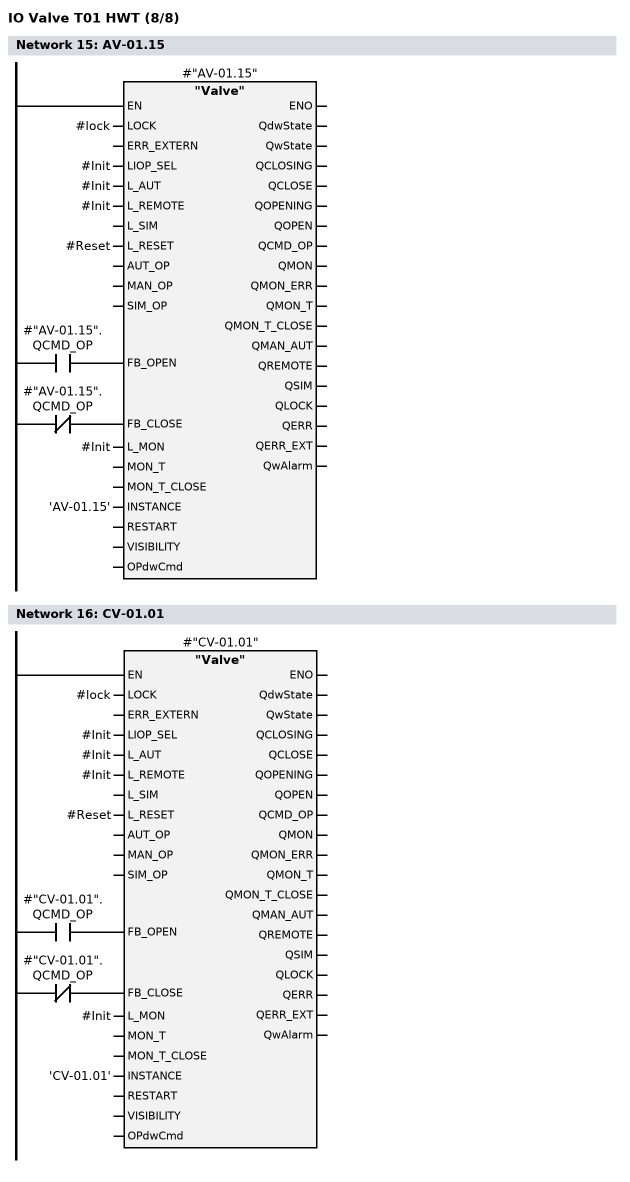
   RUNG wire#powerrail
      #"AV-01.15"(FB_OPEN := wire#w1, FB_CLOSE := wire#w2, LOCK := #lock, ERR_EXTERN :=, LIOP_SEL := #Init, L_AUT := #Init, L_REMOTE := #Init, L_SIM :=, L_RESET := #Reset, AUT_OP :=, MAN_OP :=, SIM_OP :=, L_MON := #Init, MON_T :=, MON_T_CLOSE :=, INSTANCE := 'AV-01.15', RESTART :=, VISIBILITY :=, OPdwCmd :=, QdwState =>, QwState =>, QCLOSING =>, QCLOSE =>, QOPENING =>, QOPEN =>, QCMD_OP =>, QMON =>, QMON_ERR =>, QMON_T =>, QMON_T_CLOSE =>, QMAN_AUT =>, QREMOTE =>, QSIM =>, QLOCK =>, QERR =>, QERR_EXT =>, QwAlarm =>)
   END_RUNG
   RUNG wire#powerrail
      Contact( #"AV-01.15".QCMD_OP )
   END_RUNG wire#w1
   RUNG wire#powerrail
      I_Contact( #"AV-01.15".QCMD_OP )
   END_RUNG wire#w2
   // the same network as SCL:
   #"AV-01.15"(LOCK := #lock,   // "Valve"
               LIOP_SEL := #Init,
               L_AUT := #Init,
               L_REMOTE := #Init,
               L_RESET := #Reset,
               FB_OPEN := #"AV-01.15".QCMD_OP,
               FB_CLOSE := NOT #"AV-01.15".QCMD_OP,
               L_MON := #Init,
               INSTANCE := 'AV-01.15');
END_REGION

REGION Network 16: CV-01.01
   RUNG wire#powerrail
      #"CV-01.01"(FB_OPEN := wire#w1, FB_CLOSE := wire#w2, LOCK := #lock, ERR_EXTERN :=, LIOP_SEL := #Init, L_AUT := #Init, L_REMOTE := #Init, L_SIM :=, L_RESET := #Reset, AUT_OP :=, MAN_OP :=, SIM_OP :=, L_MON := #Init, MON_T :=, MON_T_CLOSE :=, INSTANCE := 'CV-01.01', RESTART :=, VISIBILITY :=, OPdwCmd :=, QdwState =>, QwState =>, QCLOSING =>, QCLOSE =>, QOPENING =>, QOPEN =>, QCMD_OP =>, QMON =>, QMON_ERR =>, QMON_T =>, QMON_T_CLOSE =>, QMAN_AUT =>, QREMOTE =>, QSIM =>, QLOCK =>, QERR =>, QERR_EXT =>, QwAlarm =>)
   END_RUNG
   RUNG wire#powerrail
      Contact( #"CV-01.01".QCMD_OP )
   END_RUNG wire#w1
   RUNG wire#powerrail
      I_Contact( #"CV-01.01".QCMD_OP )
   END_RUNG wire#w2
   // the same network as SCL:
   #"CV-01.01"(LOCK := #lock,   // "Valve"
               LIOP_SEL := #Init,
               L_AUT := #Init,
               L_REMOTE := #Init,
               L_RESET := #Reset,
               FB_OPEN := #"CV-01.01".QCMD_OP,
               FB_CLOSE := NOT #"CV-01.01".QCMD_OP,
               L_MON := #Init,
               INSTANCE := 'CV-01.01');
END_REGION
END_FUNCTION_BLOCK

FUNCTION_BLOCK "BLEND"   // FB16, LAD
{ S7_Optimized_Access := 'FALSE' }
VERSION : 0.1
// stored: AutoNumber true, IsIECCheckEnabled false, SetENOAutomatically false, UDAEnableTagReadback false
   VAR_INPUT
      Lock : Bool := true;
      Reset : Bool;
      ENTransfer : Bool;
      ENProd : Bool;
      THE_ProdReq : Bool;   // THE Product Request
      THE_ProdLineOpen : Bool;   // THE Line Transfer Open
      THE_CIPLineOpen : Bool;   // THE CIP Line Open
      THE_CIP_En : Bool;   // THE CIP Enable
      MixproofFlip : Bool;
      FB_AV_Transfer : Bool;
      FB_P_Transfer : Bool;
      Level : Real;   // Tank Level Transmitter
      Temp : Real;   // Tank Temp Transmitter
      TransfPump_AVSpeed : Real;
   END_VAR
   VAR_OUTPUT
      Q_Prod : Bool;   // Product Available
      Q_Trans : Bool;   // Transfer to Mix in Progress
      Q_CIPReq : Bool;   // CIP Request
      Q_MixProofFlif : Bool;   // Mixproof Valve Flip
      QAV_Transfer : Bool;
      QP_Transfer : Bool;
   END_VAR
   VAR DB_SPECIFIC
      Cmd : Struct
         Transfer_ON : Bool;
         Transfer_OFF : Bool;
      END_STRUCT;
      HMI : Struct
         Cmd : DWord;
         Cmd_EN : DWord;
         Cmd_Stat : DWord;
         MatSel : DWord;
         DoseStart : DWord;
         DosePause : DWord;
         DoseStop : DWord;
         DoseState : DWord;
      END_STRUCT;
      Tank_Par : Struct
         LL : Real := 2.0;   // Tank Low Level
         LB_OFF : Real := 17.0;
         LB_ON : Real := 20.0;
         LB1_OFF : Real := 10.0;   // Level Under Lower Blade
         LB1_ON : Real := 15.0;   // Level Over Lower Blade
         LB2_OFF : Real := 30.0;   // Level Under Medium Blade
         LB2_ON : Real := 35.0;   // Level Over Medium Blade
         LB3_OFF : Real := 60.0;   // Level Under Upper Blade
         LB3_ON : Real := 65.0;   // Level Over Upper Blade
         P01_ProdSP : Real := 5.0;   // Transfer pump Setpoint speed at product transfer
         P01_CIPSP : Real := 50.0;   // Transfer pump Setpoint speed at CIP
      END_STRUCT;
      Tank_Sta : Struct   // Tank Low Level
         LL : Bool;   // Level Under Lower Blade
         LB_OFF : Bool;
         LB_ON : Bool;
         LB1_OFF : Bool;   // Level Over Lower Blade
         LB1_ON : Bool;   // Level Under Medium Blade
         LB2_OFF : Bool;   // Level Over Medium Blade
         LB2_ON : Bool;   // Level Under Upper Blade
         LB3_OFF : Bool;   // Level Over Upper Blade
         LB3_ON : Bool;
         Agi_ON : Bool;
         TranferON : Bool;
         Inload : Bool;
         CIPRequest : Bool;
         AwysON : Bool;
      END_STRUCT;
   END_VAR
   VAR
      SP_Water : "RawDose";
      SP_Sugar { S7_SetPoint := 'True'} : "RawDose";
      SP_Garam { S7_SetPoint := 'True'} : "RawDose";
      SP_ChiliAwet_1 { S7_SetPoint := 'True'} : "RawDose";
      SP_ChiliAwet_2 { S7_SetPoint := 'True'} : "RawDose";
      SP_ChiliAwet_3 { S7_SetPoint := 'True'} : "RawDose";
      SP_ChiliFresh_1 { S7_SetPoint := 'True'} : "RawDose";
      SP_ChiliFresh_2 { S7_SetPoint := 'True'} : "RawDose";
      SP_ChiliFresh_3 { S7_SetPoint := 'True'} : "RawDose";
      SP_Garlic { S7_SetPoint := 'True'} : "RawDose";
      SP_Vinegar { S7_SetPoint := 'True'} : "RawDose";
      SP_Tomato { S7_SetPoint := 'True'} : "RawDose";
      SP_Homomix { S7_SetPoint := 'True'} : "RawDose";
      SP_Rework { S7_SetPoint := 'True'} : "RawDose";
      Water : "DOSE";
      Sugar { S7_SetPoint := 'True'} : "DOSE";
      Garam : "DOSE";
      ChiliAwet_1 { S7_SetPoint := 'True'} : "DOSE";
      ChiliAwet_2 { S7_SetPoint := 'True'} : "DOSE";
      ChiliAwet_3 { S7_SetPoint := 'True'} : "DOSE";
      ChiliFresh_1 { S7_SetPoint := 'True'} : "DOSE";
      ChiliFresh_2 { S7_SetPoint := 'True'} : "DOSE";
      ChiliFresh_3 { S7_SetPoint := 'True'} : "DOSE";
      Garlic { S7_SetPoint := 'True'} : "DOSE";
      Vinegar { S7_SetPoint := 'True'} : "DOSE";
      Tomato { S7_SetPoint := 'True'} : "DOSE";
      Homomix { S7_SetPoint := 'True'} : "DOSE";
      Rework { S7_SetPoint := 'True'} : "DOSE";
   END_VAR
   VAR DB_SPECIFIC
      RdyforTransfer : Struct
         cmd_on : Bool;
         cmd_off : Bool;
         EnCmd : Bool;
         Stat_ON : Bool;
         Stat_Stop : Bool;
      END_STRUCT;
      Transfer : Struct
         cmd_on : Bool;
         cmd_off : Bool;
         EnCmd : Bool;
         Stat_ON : Bool;
         Stat_Stop : Bool;
      END_STRUCT;
      CIP : Struct
         cmd_on : Bool;
         cmd_off : Bool;
         EnCmd : Bool;
         Stat_ON : Bool;
         Stat_Stop : Bool;
      END_STRUCT;
      Agitator : Struct
         cmd_on : Bool;
         cmd_off : Bool;
         EnCmd : Bool;
         Stat_ON : Bool;
         Stat_Stop : Bool;
      END_STRUCT;
      PumpOFFTimer : TON_TIME;
      TransitionTimer { S7_SetPoint := 'True'} : TON_TIME;
   END_VAR
BEGIN

REGION Network 1: Always ON
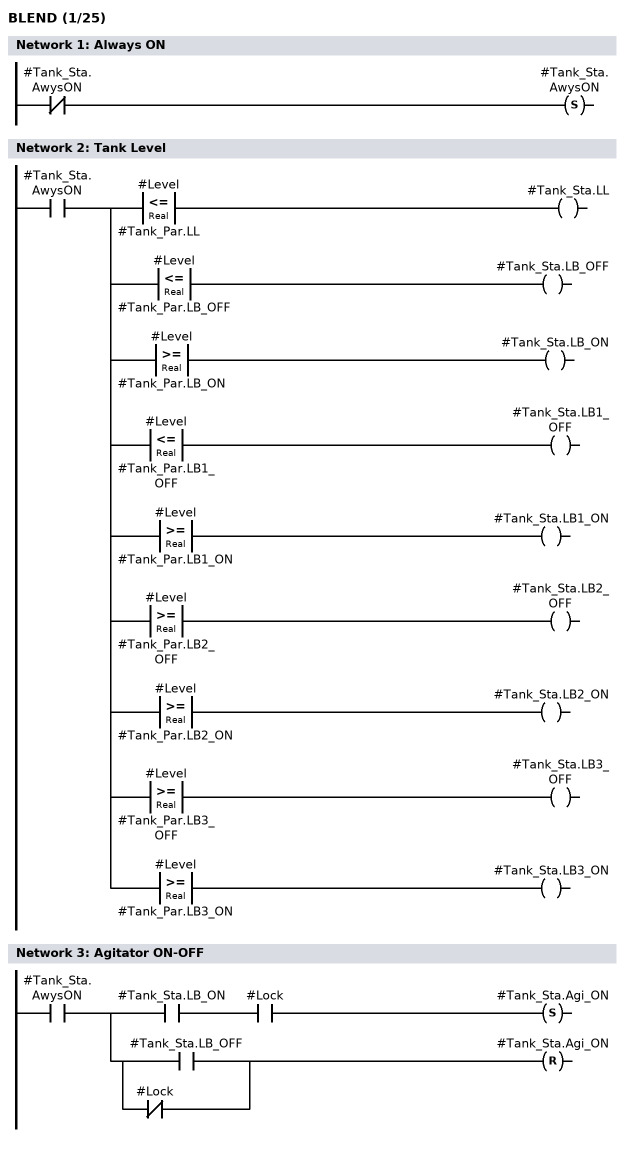
   RUNG wire#powerrail
      I_Contact( #Tank_Sta.AwysON )
      S_Coil( #Tank_Sta.AwysON )
   END_RUNG
   // the same network as SCL:
   IF NOT #Tank_Sta.AwysON THEN #Tank_Sta.AwysON := TRUE; END_IF;
END_REGION

REGION Network 2: Tank Level
   RUNG wire#powerrail
      Contact( #Tank_Sta.AwysON )
      wire#w1
      { S7_Templates := "SrcType := Real" } LE_Contact(in1 := #Level, in2 := #Tank_Par.LL)
      Coil( #Tank_Sta.LL )
   END_RUNG
   RUNG wire#w1
      { S7_Templates := "SrcType := Real" } LE_Contact(in1 := #Level, in2 := #Tank_Par.LB_OFF)
      Coil( #Tank_Sta.LB_OFF )
   END_RUNG
   RUNG wire#w1
      { S7_Templates := "SrcType := Real" } GE_Contact(in1 := #Level, in2 := #Tank_Par.LB_ON)
      Coil( #Tank_Sta.LB_ON )
   END_RUNG
   RUNG wire#w1
      { S7_Templates := "SrcType := Real" } LE_Contact(in1 := #Level, in2 := #Tank_Par.LB1_OFF)
      Coil( #Tank_Sta.LB1_OFF )
   END_RUNG
   RUNG wire#w1
      { S7_Templates := "SrcType := Real" } GE_Contact(in1 := #Level, in2 := #Tank_Par.LB1_ON)
      Coil( #Tank_Sta.LB1_ON )
   END_RUNG
   RUNG wire#w1
      { S7_Templates := "SrcType := Real" } GE_Contact(in1 := #Level, in2 := #Tank_Par.LB2_OFF)
      Coil( #Tank_Sta.LB2_OFF )
   END_RUNG
   RUNG wire#w1
      { S7_Templates := "SrcType := Real" } GE_Contact(in1 := #Level, in2 := #Tank_Par.LB2_ON)
      Coil( #Tank_Sta.LB2_ON )
   END_RUNG
   RUNG wire#w1
      { S7_Templates := "SrcType := Real" } GE_Contact(in1 := #Level, in2 := #Tank_Par.LB3_OFF)
      Coil( #Tank_Sta.LB3_OFF )
   END_RUNG
   RUNG wire#w1
      { S7_Templates := "SrcType := Real" } GE_Contact(in1 := #Level, in2 := #Tank_Par.LB3_ON)
      Coil( #Tank_Sta.LB3_ON )
   END_RUNG
   // the same network as SCL:
   #Tank_Sta.LL := #Tank_Sta.AwysON AND (#Level <= #Tank_Par.LL);
   #Tank_Sta.LB_OFF := #Tank_Sta.AwysON AND (#Level <= #Tank_Par.LB_OFF);
   #Tank_Sta.LB_ON := #Tank_Sta.AwysON AND (#Level >= #Tank_Par.LB_ON);
   #Tank_Sta.LB1_OFF := #Tank_Sta.AwysON AND (#Level <= #Tank_Par.LB1_OFF);
   #Tank_Sta.LB1_ON := #Tank_Sta.AwysON AND (#Level >= #Tank_Par.LB1_ON);
   #Tank_Sta.LB2_OFF := #Tank_Sta.AwysON AND (#Level >= #Tank_Par.LB2_OFF);
   #Tank_Sta.LB2_ON := #Tank_Sta.AwysON AND (#Level >= #Tank_Par.LB2_ON);
   #Tank_Sta.LB3_OFF := #Tank_Sta.AwysON AND (#Level >= #Tank_Par.LB3_OFF);
   #Tank_Sta.LB3_ON := #Tank_Sta.AwysON AND (#Level >= #Tank_Par.LB3_ON);
END_REGION

REGION Network 3: Agitator ON-OFF
   RUNG wire#powerrail
      Contact( #Tank_Sta.AwysON )
      wire#w1
      Contact( #Tank_Sta.LB_ON )
      Contact( #Lock )
      S_Coil( #Tank_Sta.Agi_ON )
   END_RUNG
   RUNG wire#w1
      Contact( #Tank_Sta.LB_OFF )
      wire#w2
      R_Coil( #Tank_Sta.Agi_ON )
   END_RUNG
   RUNG wire#w1
      I_Contact( #Lock )
   END_RUNG wire#w2
   // the same network as SCL:
   IF #Tank_Sta.AwysON AND #Tank_Sta.LB_ON AND #Lock THEN #Tank_Sta.Agi_ON := TRUE; END_IF;
   IF #Tank_Sta.AwysON AND (#Tank_Sta.LB_OFF OR NOT #Lock) THEN #Tank_Sta.Agi_ON := FALSE; END_IF;
END_REGION

REGION Network 5: Product Available
   // #HMI.Cmd.%X2 = Product available
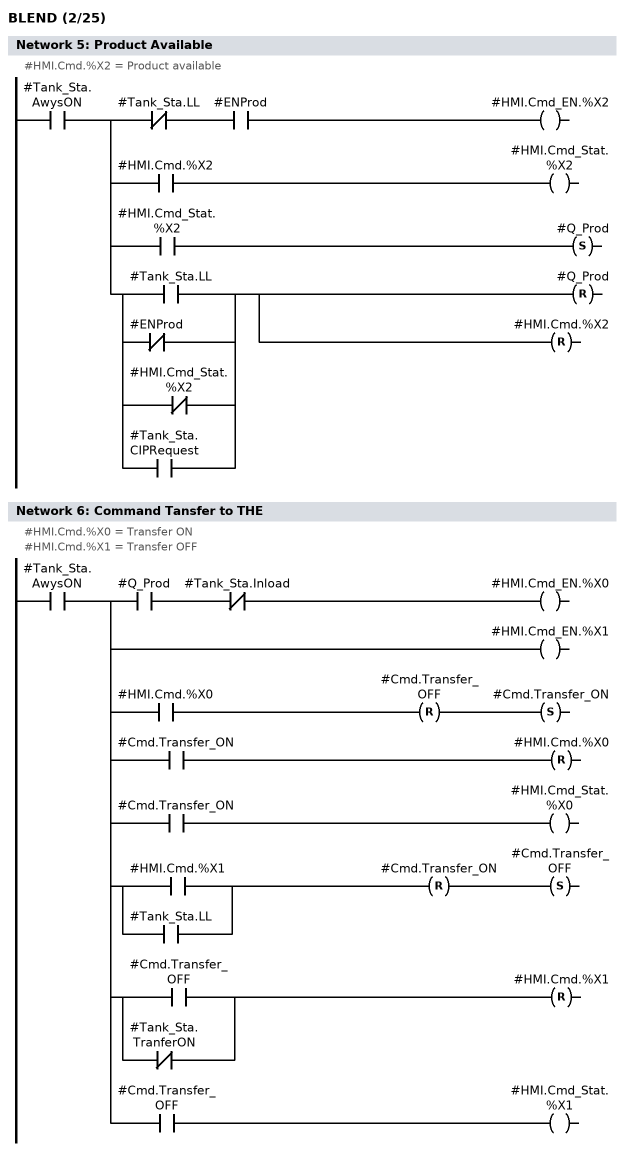
   RUNG wire#powerrail
      Contact( #Tank_Sta.AwysON )
      wire#w1
      I_Contact( #Tank_Sta.LL )
      Contact( #ENProd )
      Coil( #HMI.Cmd_EN.%X2 )
   END_RUNG
   RUNG wire#w1
      Contact( #HMI.Cmd.%X2 )
      Coil( #HMI.Cmd_Stat.%X2 )
   END_RUNG
   RUNG wire#w1
      Contact( #HMI.Cmd_Stat.%X2 )
      S_Coil( #Q_Prod )
   END_RUNG
   RUNG wire#w1
      Contact( #Tank_Sta.LL )
      wire#w2
      R_Coil( #Q_Prod )
   END_RUNG
   RUNG wire#w1
      I_Contact( #ENProd )
   END_RUNG wire#w2
   RUNG wire#w1
      I_Contact( #HMI.Cmd_Stat.%X2 )
   END_RUNG wire#w2
   RUNG wire#w1
      Contact( #Tank_Sta.CIPRequest )
   END_RUNG wire#w2
   RUNG wire#w2
      R_Coil( #HMI.Cmd.%X2 )
   END_RUNG
   // the same network as SCL:
   #HMI.Cmd_EN.%X2 := #Tank_Sta.AwysON AND NOT #Tank_Sta.LL AND #ENProd;
   #HMI.Cmd_Stat.%X2 := #Tank_Sta.AwysON AND #HMI.Cmd.%X2;
   IF #Tank_Sta.AwysON AND #HMI.Cmd_Stat.%X2 THEN #Q_Prod := TRUE; END_IF;
   IF #Tank_Sta.AwysON AND (#Tank_Sta.LL OR NOT #ENProd OR NOT #HMI.Cmd_Stat.%X2 OR #Tank_Sta.CIPRequest) THEN
       #Q_Prod := FALSE;
       #HMI.Cmd.%X2 := FALSE;
   END_IF;
END_REGION

REGION Network 6: Command Tansfer to THE
   // #HMI.Cmd.%X0 = Transfer ON
   // #HMI.Cmd.%X1 = Transfer OFF
   RUNG wire#powerrail
      Contact( #Tank_Sta.AwysON )
      wire#w1
      Contact( #Q_Prod )
      I_Contact( #Tank_Sta.Inload )
      Coil( #HMI.Cmd_EN.%X0 )
   END_RUNG
   RUNG wire#w1
      Coil( #HMI.Cmd_EN.%X1 )
   END_RUNG
   RUNG wire#w1
      Contact( #HMI.Cmd.%X0 )
      R_Coil( #Cmd.Transfer_OFF )
      S_Coil( #Cmd.Transfer_ON )
   END_RUNG
   RUNG wire#w1
      Contact( #Cmd.Transfer_ON )
      R_Coil( #HMI.Cmd.%X0 )
   END_RUNG
   RUNG wire#w1
      Contact( #Cmd.Transfer_ON )
      Coil( #HMI.Cmd_Stat.%X0 )
   END_RUNG
   RUNG wire#w1
      Contact( #HMI.Cmd.%X1 )
      wire#w2
      R_Coil( #Cmd.Transfer_ON )
      S_Coil( #Cmd.Transfer_OFF )
   END_RUNG
   RUNG wire#w1
      Contact( #Tank_Sta.LL )
   END_RUNG wire#w2
   RUNG wire#w1
      Contact( #Cmd.Transfer_OFF )
      wire#w3
      R_Coil( #HMI.Cmd.%X1 )
   END_RUNG
   RUNG wire#w1
      I_Contact( #Tank_Sta.TranferON )
   END_RUNG wire#w3
   RUNG wire#w1
      Contact( #Cmd.Transfer_OFF )
      Coil( #HMI.Cmd_Stat.%X1 )
   END_RUNG
   // the same network as SCL:
   #HMI.Cmd_EN.%X0 := #Tank_Sta.AwysON AND #Q_Prod AND NOT #Tank_Sta.Inload;
   #HMI.Cmd_EN.%X1 := #Tank_Sta.AwysON;
   IF #Tank_Sta.AwysON AND #HMI.Cmd.%X0 THEN
       #Cmd.Transfer_OFF := FALSE;
       #Cmd.Transfer_ON := TRUE;
   END_IF;
   IF #Tank_Sta.AwysON AND #Cmd.Transfer_ON THEN #HMI.Cmd.%X0 := FALSE; END_IF;
   #HMI.Cmd_Stat.%X0 := #Tank_Sta.AwysON AND #Cmd.Transfer_ON;
   IF #Tank_Sta.AwysON AND (#HMI.Cmd.%X1 OR #Tank_Sta.LL) THEN
       #Cmd.Transfer_ON := FALSE;
       #Cmd.Transfer_OFF := TRUE;
   END_IF;
   IF #Tank_Sta.AwysON AND (#Cmd.Transfer_OFF OR NOT #Tank_Sta.TranferON) THEN #HMI.Cmd.%X1 := FALSE; END_IF;
   #HMI.Cmd_Stat.%X1 := #Tank_Sta.AwysON AND #Cmd.Transfer_OFF;
END_REGION

REGION Network 7: Tansfer to THE
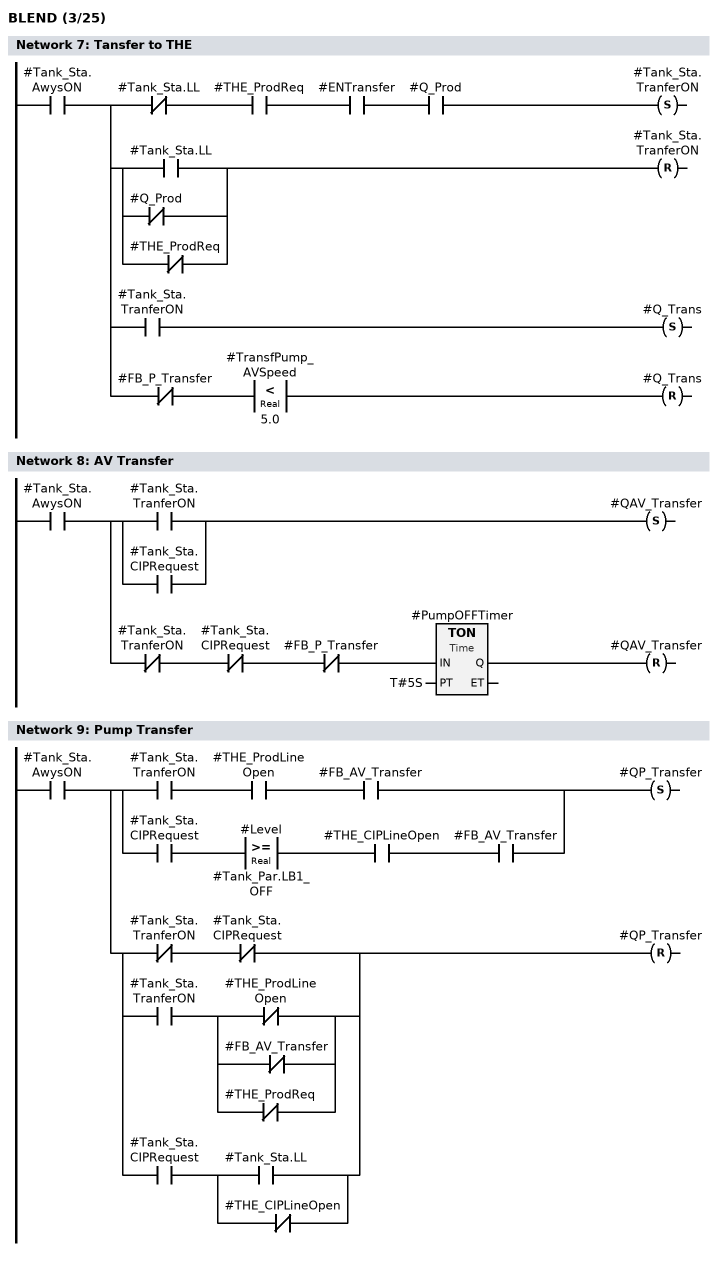
   RUNG wire#powerrail
      Contact( #Tank_Sta.AwysON )
      wire#w1
      I_Contact( #Tank_Sta.LL )
      Contact( #THE_ProdReq )
      Contact( #ENTransfer )
      Contact( #Q_Prod )
      S_Coil( #Tank_Sta.TranferON )
   END_RUNG
   RUNG wire#w1
      Contact( #Tank_Sta.LL )
      wire#w2
      R_Coil( #Tank_Sta.TranferON )
   END_RUNG
   RUNG wire#w1
      I_Contact( #Q_Prod )
   END_RUNG wire#w2
   RUNG wire#w1
      I_Contact( #THE_ProdReq )
   END_RUNG wire#w2
   RUNG wire#w1
      Contact( #Tank_Sta.TranferON )
      S_Coil( #Q_Trans )
   END_RUNG
   RUNG wire#w1
      I_Contact( #FB_P_Transfer )
      { S7_Templates := "SrcType := Real" } LT_Contact(in1 := #TransfPump_AVSpeed, in2 := 5.0)
      R_Coil( #Q_Trans )
   END_RUNG
   // the same network as SCL:
   IF #Tank_Sta.AwysON AND NOT #Tank_Sta.LL AND #THE_ProdReq AND #ENTransfer AND #Q_Prod THEN
       #Tank_Sta.TranferON := TRUE;
   END_IF;
   IF #Tank_Sta.AwysON AND (#Tank_Sta.LL OR NOT #Q_Prod OR NOT #THE_ProdReq) THEN
       #Tank_Sta.TranferON := FALSE;
   END_IF;
   IF #Tank_Sta.AwysON AND #Tank_Sta.TranferON THEN #Q_Trans := TRUE; END_IF;
   IF #Tank_Sta.AwysON AND NOT #FB_P_Transfer AND (#TransfPump_AVSpeed < 5.0) THEN #Q_Trans := FALSE; END_IF;
END_REGION

REGION Network 8: AV Transfer
   RUNG wire#powerrail
      Contact( #Tank_Sta.AwysON )
      wire#w1
      Contact( #Tank_Sta.TranferON )
      wire#w2
      S_Coil( #QAV_Transfer )
   END_RUNG
   RUNG wire#w1
      Contact( #Tank_Sta.CIPRequest )
   END_RUNG wire#w2
   RUNG wire#w1
      I_Contact( #Tank_Sta.TranferON )
      I_Contact( #Tank_Sta.CIPRequest )
      I_Contact( #FB_P_Transfer )
      { S7_Templates := "time_type := Time" } #PumpOFFTimer.TON(pt := T#5S, et =>)
      R_Coil( #QAV_Transfer )
   END_RUNG
   // the same network as SCL:
   IF #Tank_Sta.AwysON AND (#Tank_Sta.TranferON OR #Tank_Sta.CIPRequest) THEN #QAV_Transfer := TRUE; END_IF;
   #PumpOFFTimer(IN := #Tank_Sta.AwysON AND NOT #Tank_Sta.TranferON AND NOT #Tank_Sta.CIPRequest AND NOT #FB_P_Transfer,   // TON
                 PT := T#5S);
   IF #PumpOFFTimer.Q THEN #QAV_Transfer := FALSE; END_IF;
END_REGION

REGION Network 9: Pump Transfer
   RUNG wire#powerrail
      Contact( #Tank_Sta.AwysON )
      wire#w1
      Contact( #Tank_Sta.TranferON )
      Contact( #THE_ProdLineOpen )
      Contact( #FB_AV_Transfer )
      wire#w2
      S_Coil( #QP_Transfer )
   END_RUNG
   RUNG wire#w1
      Contact( #Tank_Sta.CIPRequest )
      { S7_Templates := "SrcType := Real" } GE_Contact(in1 := #Level, in2 := #Tank_Par.LB1_OFF)
      Contact( #THE_CIPLineOpen )
      Contact( #FB_AV_Transfer )
   END_RUNG wire#w2
   RUNG wire#w1
      I_Contact( #Tank_Sta.TranferON )
      I_Contact( #Tank_Sta.CIPRequest )
      wire#w3
      R_Coil( #QP_Transfer )
   END_RUNG
   RUNG wire#w1
      Contact( #Tank_Sta.TranferON )
      wire#w4
      I_Contact( #THE_ProdLineOpen )
   END_RUNG wire#w3
   RUNG wire#w4
      I_Contact( #FB_AV_Transfer )
   END_RUNG wire#w3
   RUNG wire#w4
      I_Contact( #THE_ProdReq )
   END_RUNG wire#w3
   RUNG wire#w1
      Contact( #Tank_Sta.CIPRequest )
      wire#w5
      Contact( #Tank_Sta.LL )
   END_RUNG wire#w3
   RUNG wire#w5
      I_Contact( #THE_CIPLineOpen )
   END_RUNG wire#w3
   // the same network as SCL:
   IF #Tank_Sta.AwysON AND ((#Tank_Sta.TranferON AND #THE_ProdLineOpen AND #FB_AV_Transfer) OR (#Tank_Sta.CIPRequest AND (#Level >= #Tank_Par.LB1_OFF) AND #THE_CIPLineOpen AND #FB_AV_Transfer)) THEN
       #QP_Transfer := TRUE;
   END_IF;
   IF #Tank_Sta.AwysON AND ((NOT #Tank_Sta.TranferON AND NOT #Tank_Sta.CIPRequest) OR (#Tank_Sta.TranferON AND (NOT #THE_ProdLineOpen OR NOT #FB_AV_Transfer OR NOT #THE_ProdReq)) OR (#Tank_Sta.CIPRequest AND (#Tank_Sta.LL OR NOT #THE_CIPLineOpen))) THEN
       #QP_Transfer := FALSE;
   END_IF;
END_REGION

REGION Network 10: CIP Request
   // #HMI.Cmd.%X4 = CIP Request ON
   // #HMI.Cmd.%X5 = CIP Request OFF
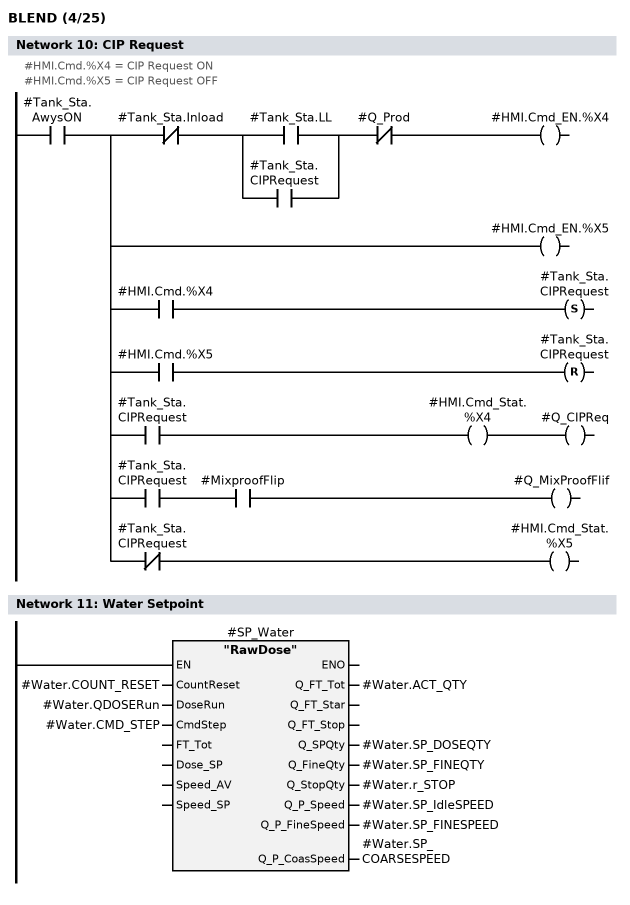
   RUNG wire#powerrail
      Contact( #Tank_Sta.AwysON )
      wire#w1
      I_Contact( #Tank_Sta.Inload )
      wire#w2
      Contact( #Tank_Sta.LL )
      wire#w3
      I_Contact( #Q_Prod )
      Coil( #HMI.Cmd_EN.%X4 )
   END_RUNG
   RUNG wire#w2
      Contact( #Tank_Sta.CIPRequest )
   END_RUNG wire#w3
   RUNG wire#w1
      Coil( #HMI.Cmd_EN.%X5 )
   END_RUNG
   RUNG wire#w1
      Contact( #HMI.Cmd.%X4 )
      S_Coil( #Tank_Sta.CIPRequest )
   END_RUNG
   RUNG wire#w1
      Contact( #HMI.Cmd.%X5 )
      R_Coil( #Tank_Sta.CIPRequest )
   END_RUNG
   RUNG wire#w1
      Contact( #Tank_Sta.CIPRequest )
      Coil( #HMI.Cmd_Stat.%X4 )
      Coil( #Q_CIPReq )
   END_RUNG
   RUNG wire#w1
      Contact( #Tank_Sta.CIPRequest )
      Contact( #MixproofFlip )
      Coil( #Q_MixProofFlif )
   END_RUNG
   RUNG wire#w1
      I_Contact( #Tank_Sta.CIPRequest )
      Coil( #HMI.Cmd_Stat.%X5 )
   END_RUNG
   // the same network as SCL:
   #HMI.Cmd_EN.%X4 := #Tank_Sta.AwysON AND NOT #Tank_Sta.Inload AND (#Tank_Sta.LL OR #Tank_Sta.CIPRequest) AND NOT #Q_Prod;
   #HMI.Cmd_EN.%X5 := #Tank_Sta.AwysON;
   IF #Tank_Sta.AwysON AND #HMI.Cmd.%X4 THEN #Tank_Sta.CIPRequest := TRUE; END_IF;
   IF #Tank_Sta.AwysON AND #HMI.Cmd.%X5 THEN #Tank_Sta.CIPRequest := FALSE; END_IF;
   #HMI.Cmd_Stat.%X4 := #Tank_Sta.AwysON AND #Tank_Sta.CIPRequest;
   #Q_CIPReq := #HMI.Cmd_Stat.%X4;
   #Q_MixProofFlif := #Tank_Sta.AwysON AND #Tank_Sta.CIPRequest AND #MixproofFlip;
   #HMI.Cmd_Stat.%X5 := #Tank_Sta.AwysON AND NOT #Tank_Sta.CIPRequest;
END_REGION

REGION Network 11: Water Setpoint
   RUNG wire#powerrail
      #SP_Water(CountReset := #Water.COUNT_RESET, DoseRun := #Water.QDOSERun, CmdStep := #Water.CMD_STEP, FT_Tot :=, Dose_SP :=, Speed_AV :=, Speed_SP :=, Q_FT_Tot => #Water.ACT_QTY, Q_FT_Star =>, Q_FT_Stop =>, Q_SPQty => #Water.SP_DOSEQTY, Q_FineQty => #Water.SP_FINEQTY, Q_StopQty => #Water.r_STOP, Q_P_Speed => #Water.SP_IdleSPEED, Q_P_FineSpeed => #Water.SP_FINESPEED, Q_P_CoasSpeed => #Water.SP_COARSESPEED)
   END_RUNG
   // the same network as SCL:
   #SP_Water(CountReset := #Water.COUNT_RESET,   // "RawDose"
             DoseRun := #Water.QDOSERun,
             CmdStep := #Water.CMD_STEP,
             Q_FT_Tot => #Water.ACT_QTY,
             Q_SPQty => #Water.SP_DOSEQTY,
             Q_FineQty => #Water.SP_FINEQTY,
             Q_StopQty => #Water.r_STOP,
             Q_P_Speed => #Water.SP_IdleSPEED,
             Q_P_FineSpeed => #Water.SP_FINESPEED,
             Q_P_CoasSpeed => #Water.SP_COARSESPEED);
END_REGION

REGION Network 12: Dose Water
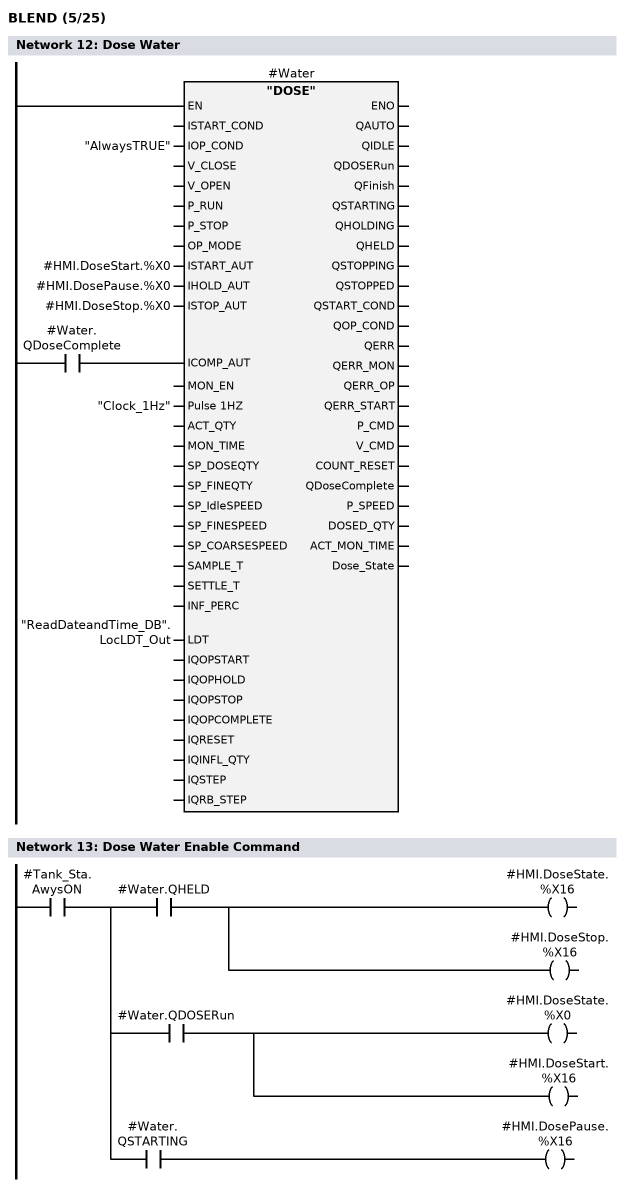
   RUNG wire#powerrail
      #Water(ICOMP_AUT := wire#w1, ISTART_COND :=, IOP_COND := "AlwaysTRUE", V_CLOSE :=, V_OPEN :=, P_RUN :=, P_STOP :=, OP_MODE :=, ISTART_AUT := #HMI.DoseStart.%X0, IHOLD_AUT := #HMI.DosePause.%X0, ISTOP_AUT := #HMI.DoseStop.%X0, MON_EN :=, "Pulse 1HZ" := "Clock_1Hz", ACT_QTY :=, MON_TIME :=, SP_DOSEQTY :=, SP_FINEQTY :=, SP_IdleSPEED :=, SP_FINESPEED :=, SP_COARSESPEED :=, SAMPLE_T :=, SETTLE_T :=, INF_PERC :=, LDT := "ReadDateandTime_DB".LocLDT_Out, IQOPSTART :=, IQOPHOLD :=, IQOPSTOP :=, IQOPCOMPLETE :=, IQRESET :=, IQINFL_QTY :=, IQSTEP :=, IQRB_STEP :=, QAUTO =>, QIDLE =>, QDOSERun =>, QFinish =>, QSTARTING =>, QHOLDING =>, QHELD =>, QSTOPPING =>, QSTOPPED =>, QSTART_COND =>, QOP_COND =>, QERR =>, QERR_MON =>, QERR_OP =>, QERR_START =>, P_CMD =>, V_CMD =>, COUNT_RESET =>, QDoseComplete =>, P_SPEED =>, DOSED_QTY =>, ACT_MON_TIME =>, Dose_State =>)
   END_RUNG
   RUNG wire#powerrail
      Contact( #Water.QDoseComplete )
   END_RUNG wire#w1
   // the same network as SCL:
   #Water(IOP_COND := "AlwaysTRUE",   // "DOSE"
          ISTART_AUT := #HMI.DoseStart.%X0,
          IHOLD_AUT := #HMI.DosePause.%X0,
          ISTOP_AUT := #HMI.DoseStop.%X0,
          ICOMP_AUT := #Water.QDoseComplete,
          "Pulse 1HZ" := "Clock_1Hz",
          LDT := "ReadDateandTime_DB".LocLDT_Out);
END_REGION

REGION Network 13: Dose Water Enable Command
   RUNG wire#powerrail
      Contact( #Tank_Sta.AwysON )
      wire#w1
      Contact( #Water.QHELD )
      wire#w2
      Coil( #HMI.DoseState.%X16 )
   END_RUNG
   RUNG wire#w2
      Coil( #HMI.DoseStop.%X16 )
   END_RUNG
   RUNG wire#w1
      Contact( #Water.QDOSERun )
      wire#w3
      Coil( #HMI.DoseState.%X0 )
   END_RUNG
   RUNG wire#w3
      Coil( #HMI.DoseStart.%X16 )
   END_RUNG
   RUNG wire#w1
      Contact( #Water.QSTARTING )
      Coil( #HMI.DosePause.%X16 )
   END_RUNG
   // the same network as SCL:
   #HMI.DoseState.%X16 := #Tank_Sta.AwysON AND #Water.QHELD;
   #HMI.DoseStop.%X16 := #HMI.DoseState.%X16;
   #HMI.DoseState.%X0 := #Tank_Sta.AwysON AND #Water.QDOSERun;
   #HMI.DoseStart.%X16 := #HMI.DoseState.%X0;
   #HMI.DosePause.%X16 := #Tank_Sta.AwysON AND #Water.QSTARTING;
END_REGION

REGION Network 15: Sugar Setpoint
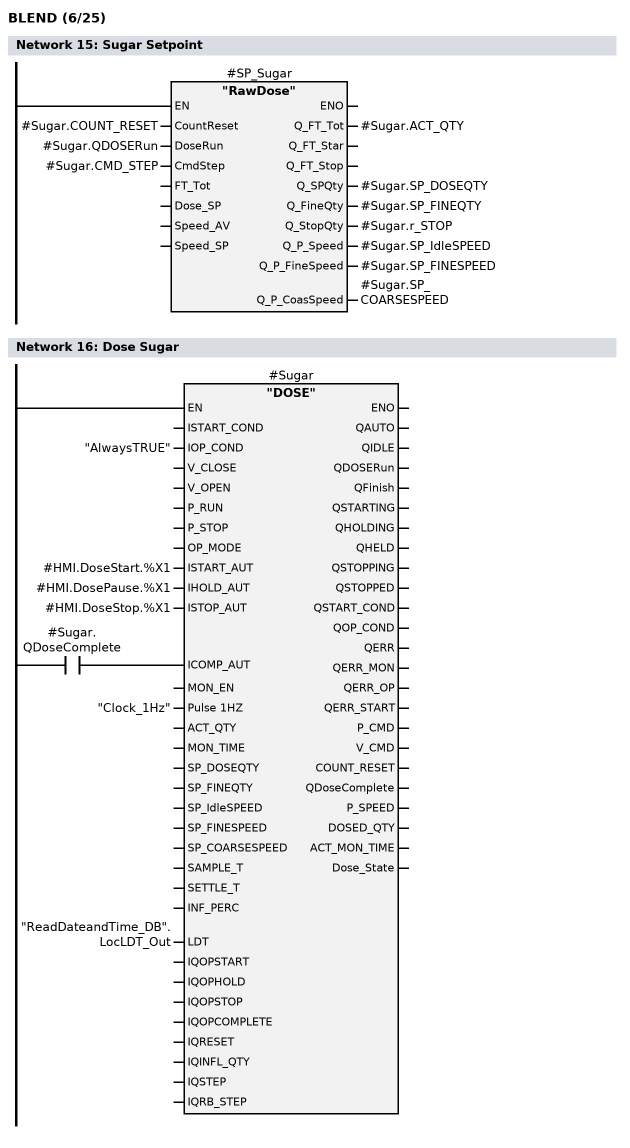
   RUNG wire#powerrail
      #SP_Sugar(CountReset := #Sugar.COUNT_RESET, DoseRun := #Sugar.QDOSERun, CmdStep := #Sugar.CMD_STEP, FT_Tot :=, Dose_SP :=, Speed_AV :=, Speed_SP :=, Q_FT_Tot => #Sugar.ACT_QTY, Q_FT_Star =>, Q_FT_Stop =>, Q_SPQty => #Sugar.SP_DOSEQTY, Q_FineQty => #Sugar.SP_FINEQTY, Q_StopQty => #Sugar.r_STOP, Q_P_Speed => #Sugar.SP_IdleSPEED, Q_P_FineSpeed => #Sugar.SP_FINESPEED, Q_P_CoasSpeed => #Sugar.SP_COARSESPEED)
   END_RUNG
   // the same network as SCL:
   #SP_Sugar(CountReset := #Sugar.COUNT_RESET,   // "RawDose"
             DoseRun := #Sugar.QDOSERun,
             CmdStep := #Sugar.CMD_STEP,
             Q_FT_Tot => #Sugar.ACT_QTY,
             Q_SPQty => #Sugar.SP_DOSEQTY,
             Q_FineQty => #Sugar.SP_FINEQTY,
             Q_StopQty => #Sugar.r_STOP,
             Q_P_Speed => #Sugar.SP_IdleSPEED,
             Q_P_FineSpeed => #Sugar.SP_FINESPEED,
             Q_P_CoasSpeed => #Sugar.SP_COARSESPEED);
END_REGION

REGION Network 16: Dose Sugar
   RUNG wire#powerrail
      #Sugar(ICOMP_AUT := wire#w1, ISTART_COND :=, IOP_COND := "AlwaysTRUE", V_CLOSE :=, V_OPEN :=, P_RUN :=, P_STOP :=, OP_MODE :=, ISTART_AUT := #HMI.DoseStart.%X1, IHOLD_AUT := #HMI.DosePause.%X1, ISTOP_AUT := #HMI.DoseStop.%X1, MON_EN :=, "Pulse 1HZ" := "Clock_1Hz", ACT_QTY :=, MON_TIME :=, SP_DOSEQTY :=, SP_FINEQTY :=, SP_IdleSPEED :=, SP_FINESPEED :=, SP_COARSESPEED :=, SAMPLE_T :=, SETTLE_T :=, INF_PERC :=, LDT := "ReadDateandTime_DB".LocLDT_Out, IQOPSTART :=, IQOPHOLD :=, IQOPSTOP :=, IQOPCOMPLETE :=, IQRESET :=, IQINFL_QTY :=, IQSTEP :=, IQRB_STEP :=, QAUTO =>, QIDLE =>, QDOSERun =>, QFinish =>, QSTARTING =>, QHOLDING =>, QHELD =>, QSTOPPING =>, QSTOPPED =>, QSTART_COND =>, QOP_COND =>, QERR =>, QERR_MON =>, QERR_OP =>, QERR_START =>, P_CMD =>, V_CMD =>, COUNT_RESET =>, QDoseComplete =>, P_SPEED =>, DOSED_QTY =>, ACT_MON_TIME =>, Dose_State =>)
   END_RUNG
   RUNG wire#powerrail
      Contact( #Sugar.QDoseComplete )
   END_RUNG wire#w1
   // the same network as SCL:
   #Sugar(IOP_COND := "AlwaysTRUE",   // "DOSE"
          ISTART_AUT := #HMI.DoseStart.%X1,
          IHOLD_AUT := #HMI.DosePause.%X1,
          ISTOP_AUT := #HMI.DoseStop.%X1,
          ICOMP_AUT := #Sugar.QDoseComplete,
          "Pulse 1HZ" := "Clock_1Hz",
          LDT := "ReadDateandTime_DB".LocLDT_Out);
END_REGION

REGION Network 17: Dose Sugar Enable Command
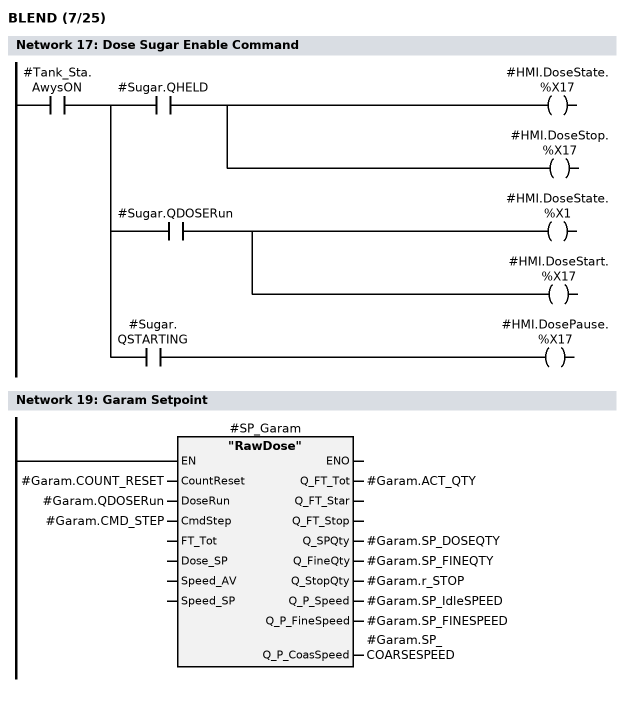
   RUNG wire#powerrail
      Contact( #Tank_Sta.AwysON )
      wire#w1
      Contact( #Sugar.QHELD )
      wire#w2
      Coil( #HMI.DoseState.%X17 )
   END_RUNG
   RUNG wire#w2
      Coil( #HMI.DoseStop.%X17 )
   END_RUNG
   RUNG wire#w1
      Contact( #Sugar.QDOSERun )
      wire#w3
      Coil( #HMI.DoseState.%X1 )
   END_RUNG
   RUNG wire#w3
      Coil( #HMI.DoseStart.%X17 )
   END_RUNG
   RUNG wire#w1
      Contact( #Sugar.QSTARTING )
      Coil( #HMI.DosePause.%X17 )
   END_RUNG
   // the same network as SCL:
   #HMI.DoseState.%X17 := #Tank_Sta.AwysON AND #Sugar.QHELD;
   #HMI.DoseStop.%X17 := #HMI.DoseState.%X17;
   #HMI.DoseState.%X1 := #Tank_Sta.AwysON AND #Sugar.QDOSERun;
   #HMI.DoseStart.%X17 := #HMI.DoseState.%X1;
   #HMI.DosePause.%X17 := #Tank_Sta.AwysON AND #Sugar.QSTARTING;
END_REGION

REGION Network 19: Garam Setpoint
   RUNG wire#powerrail
      #SP_Garam(CountReset := #Garam.COUNT_RESET, DoseRun := #Garam.QDOSERun, CmdStep := #Garam.CMD_STEP, FT_Tot :=, Dose_SP :=, Speed_AV :=, Speed_SP :=, Q_FT_Tot => #Garam.ACT_QTY, Q_FT_Star =>, Q_FT_Stop =>, Q_SPQty => #Garam.SP_DOSEQTY, Q_FineQty => #Garam.SP_FINEQTY, Q_StopQty => #Garam.r_STOP, Q_P_Speed => #Garam.SP_IdleSPEED, Q_P_FineSpeed => #Garam.SP_FINESPEED, Q_P_CoasSpeed => #Garam.SP_COARSESPEED)
   END_RUNG
   // the same network as SCL:
   #SP_Garam(CountReset := #Garam.COUNT_RESET,   // "RawDose"
             DoseRun := #Garam.QDOSERun,
             CmdStep := #Garam.CMD_STEP,
             Q_FT_Tot => #Garam.ACT_QTY,
             Q_SPQty => #Garam.SP_DOSEQTY,
             Q_FineQty => #Garam.SP_FINEQTY,
             Q_StopQty => #Garam.r_STOP,
             Q_P_Speed => #Garam.SP_IdleSPEED,
             Q_P_FineSpeed => #Garam.SP_FINESPEED,
             Q_P_CoasSpeed => #Garam.SP_COARSESPEED);
END_REGION

REGION Network 20: Dose Garam
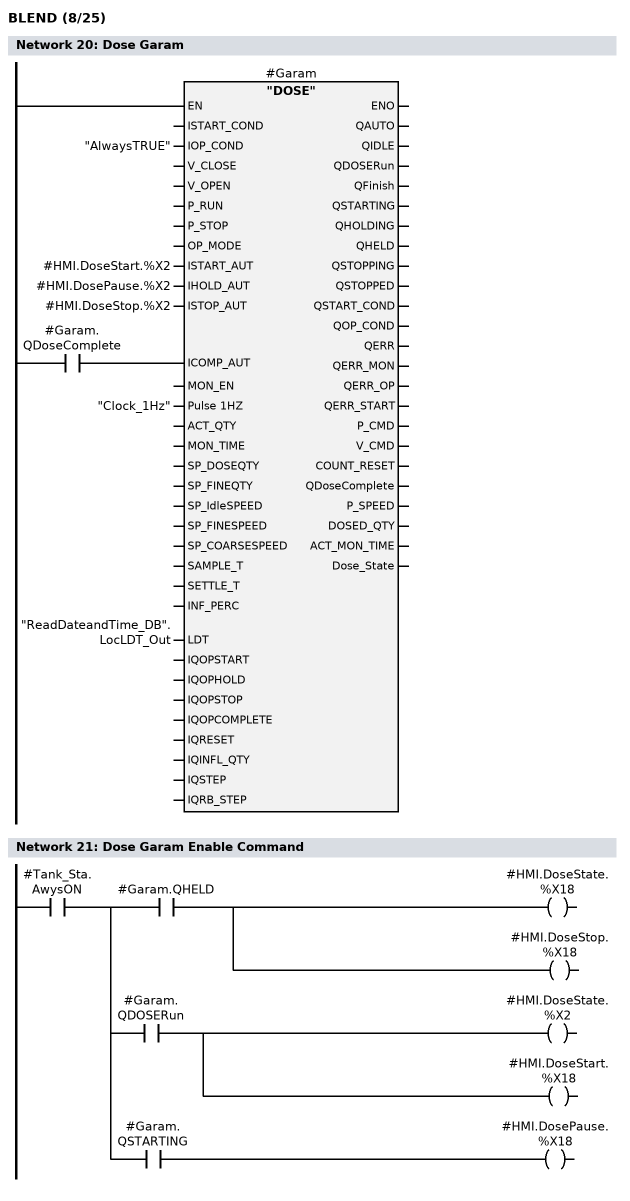
   RUNG wire#powerrail
      #Garam(ICOMP_AUT := wire#w1, ISTART_COND :=, IOP_COND := "AlwaysTRUE", V_CLOSE :=, V_OPEN :=, P_RUN :=, P_STOP :=, OP_MODE :=, ISTART_AUT := #HMI.DoseStart.%X2, IHOLD_AUT := #HMI.DosePause.%X2, ISTOP_AUT := #HMI.DoseStop.%X2, MON_EN :=, "Pulse 1HZ" := "Clock_1Hz", ACT_QTY :=, MON_TIME :=, SP_DOSEQTY :=, SP_FINEQTY :=, SP_IdleSPEED :=, SP_FINESPEED :=, SP_COARSESPEED :=, SAMPLE_T :=, SETTLE_T :=, INF_PERC :=, LDT := "ReadDateandTime_DB".LocLDT_Out, IQOPSTART :=, IQOPHOLD :=, IQOPSTOP :=, IQOPCOMPLETE :=, IQRESET :=, IQINFL_QTY :=, IQSTEP :=, IQRB_STEP :=, QAUTO =>, QIDLE =>, QDOSERun =>, QFinish =>, QSTARTING =>, QHOLDING =>, QHELD =>, QSTOPPING =>, QSTOPPED =>, QSTART_COND =>, QOP_COND =>, QERR =>, QERR_MON =>, QERR_OP =>, QERR_START =>, P_CMD =>, V_CMD =>, COUNT_RESET =>, QDoseComplete =>, P_SPEED =>, DOSED_QTY =>, ACT_MON_TIME =>, Dose_State =>)
   END_RUNG
   RUNG wire#powerrail
      Contact( #Garam.QDoseComplete )
   END_RUNG wire#w1
   // the same network as SCL:
   #Garam(IOP_COND := "AlwaysTRUE",   // "DOSE"
          ISTART_AUT := #HMI.DoseStart.%X2,
          IHOLD_AUT := #HMI.DosePause.%X2,
          ISTOP_AUT := #HMI.DoseStop.%X2,
          ICOMP_AUT := #Garam.QDoseComplete,
          "Pulse 1HZ" := "Clock_1Hz",
          LDT := "ReadDateandTime_DB".LocLDT_Out);
END_REGION

REGION Network 21: Dose Garam Enable Command
   RUNG wire#powerrail
      Contact( #Tank_Sta.AwysON )
      wire#w1
      Contact( #Garam.QHELD )
      wire#w2
      Coil( #HMI.DoseState.%X18 )
   END_RUNG
   RUNG wire#w2
      Coil( #HMI.DoseStop.%X18 )
   END_RUNG
   RUNG wire#w1
      Contact( #Garam.QDOSERun )
      wire#w3
      Coil( #HMI.DoseState.%X2 )
   END_RUNG
   RUNG wire#w3
      Coil( #HMI.DoseStart.%X18 )
   END_RUNG
   RUNG wire#w1
      Contact( #Garam.QSTARTING )
      Coil( #HMI.DosePause.%X18 )
   END_RUNG
   // the same network as SCL:
   #HMI.DoseState.%X18 := #Tank_Sta.AwysON AND #Garam.QHELD;
   #HMI.DoseStop.%X18 := #HMI.DoseState.%X18;
   #HMI.DoseState.%X2 := #Tank_Sta.AwysON AND #Garam.QDOSERun;
   #HMI.DoseStart.%X18 := #HMI.DoseState.%X2;
   #HMI.DosePause.%X18 := #Tank_Sta.AwysON AND #Garam.QSTARTING;
END_REGION

REGION Network 23: ChiliAwet_1 Setpoint
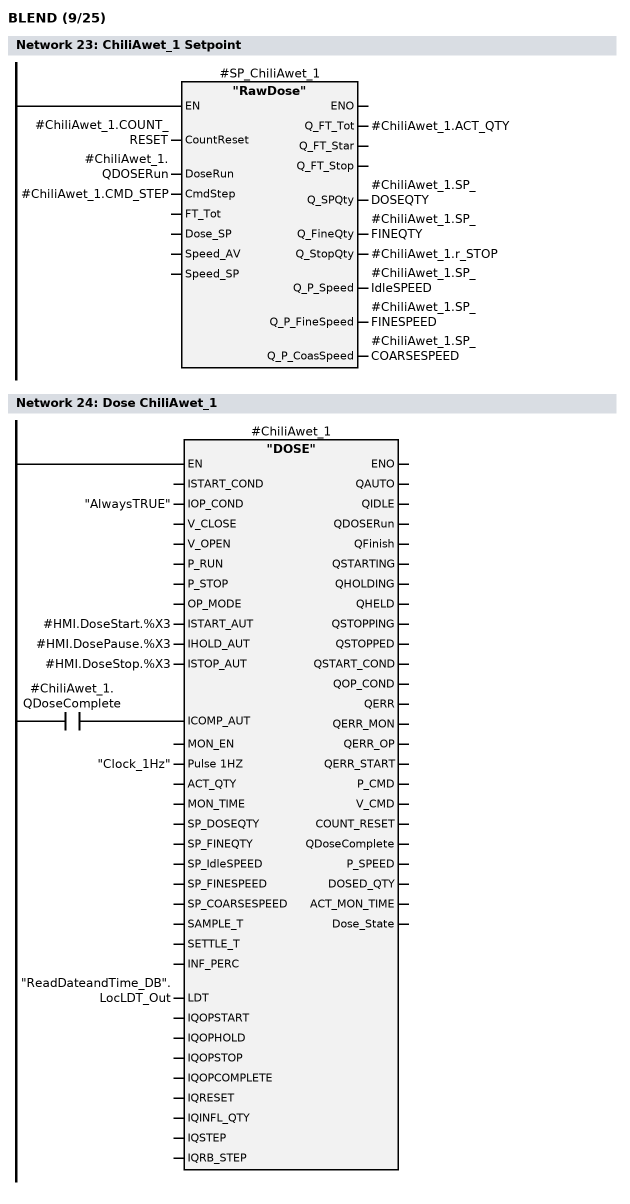
   RUNG wire#powerrail
      #SP_ChiliAwet_1(CountReset := #ChiliAwet_1.COUNT_RESET, DoseRun := #ChiliAwet_1.QDOSERun, CmdStep := #ChiliAwet_1.CMD_STEP, FT_Tot :=, Dose_SP :=, Speed_AV :=, Speed_SP :=, Q_FT_Tot => #ChiliAwet_1.ACT_QTY, Q_FT_Star =>, Q_FT_Stop =>, Q_SPQty => #ChiliAwet_1.SP_DOSEQTY, Q_FineQty => #ChiliAwet_1.SP_FINEQTY, Q_StopQty => #ChiliAwet_1.r_STOP, Q_P_Speed => #ChiliAwet_1.SP_IdleSPEED, Q_P_FineSpeed => #ChiliAwet_1.SP_FINESPEED, Q_P_CoasSpeed => #ChiliAwet_1.SP_COARSESPEED)
   END_RUNG
   // the same network as SCL:
   #SP_ChiliAwet_1(CountReset := #ChiliAwet_1.COUNT_RESET,   // "RawDose"
                   DoseRun := #ChiliAwet_1.QDOSERun,
                   CmdStep := #ChiliAwet_1.CMD_STEP,
                   Q_FT_Tot => #ChiliAwet_1.ACT_QTY,
                   Q_SPQty => #ChiliAwet_1.SP_DOSEQTY,
                   Q_FineQty => #ChiliAwet_1.SP_FINEQTY,
                   Q_StopQty => #ChiliAwet_1.r_STOP,
                   Q_P_Speed => #ChiliAwet_1.SP_IdleSPEED,
                   Q_P_FineSpeed => #ChiliAwet_1.SP_FINESPEED,
                   Q_P_CoasSpeed => #ChiliAwet_1.SP_COARSESPEED);
END_REGION

REGION Network 24: Dose ChiliAwet_1
   RUNG wire#powerrail
      #ChiliAwet_1(ICOMP_AUT := wire#w1, ISTART_COND :=, IOP_COND := "AlwaysTRUE", V_CLOSE :=, V_OPEN :=, P_RUN :=, P_STOP :=, OP_MODE :=, ISTART_AUT := #HMI.DoseStart.%X3, IHOLD_AUT := #HMI.DosePause.%X3, ISTOP_AUT := #HMI.DoseStop.%X3, MON_EN :=, "Pulse 1HZ" := "Clock_1Hz", ACT_QTY :=, MON_TIME :=, SP_DOSEQTY :=, SP_FINEQTY :=, SP_IdleSPEED :=, SP_FINESPEED :=, SP_COARSESPEED :=, SAMPLE_T :=, SETTLE_T :=, INF_PERC :=, LDT := "ReadDateandTime_DB".LocLDT_Out, IQOPSTART :=, IQOPHOLD :=, IQOPSTOP :=, IQOPCOMPLETE :=, IQRESET :=, IQINFL_QTY :=, IQSTEP :=, IQRB_STEP :=, QAUTO =>, QIDLE =>, QDOSERun =>, QFinish =>, QSTARTING =>, QHOLDING =>, QHELD =>, QSTOPPING =>, QSTOPPED =>, QSTART_COND =>, QOP_COND =>, QERR =>, QERR_MON =>, QERR_OP =>, QERR_START =>, P_CMD =>, V_CMD =>, COUNT_RESET =>, QDoseComplete =>, P_SPEED =>, DOSED_QTY =>, ACT_MON_TIME =>, Dose_State =>)
   END_RUNG
   RUNG wire#powerrail
      Contact( #ChiliAwet_1.QDoseComplete )
   END_RUNG wire#w1
   // the same network as SCL:
   #ChiliAwet_1(IOP_COND := "AlwaysTRUE",   // "DOSE"
                ISTART_AUT := #HMI.DoseStart.%X3,
                IHOLD_AUT := #HMI.DosePause.%X3,
                ISTOP_AUT := #HMI.DoseStop.%X3,
                ICOMP_AUT := #ChiliAwet_1.QDoseComplete,
                "Pulse 1HZ" := "Clock_1Hz",
                LDT := "ReadDateandTime_DB".LocLDT_Out);
END_REGION

REGION Network 25: Dose ChiliAwet_1 Enable Command
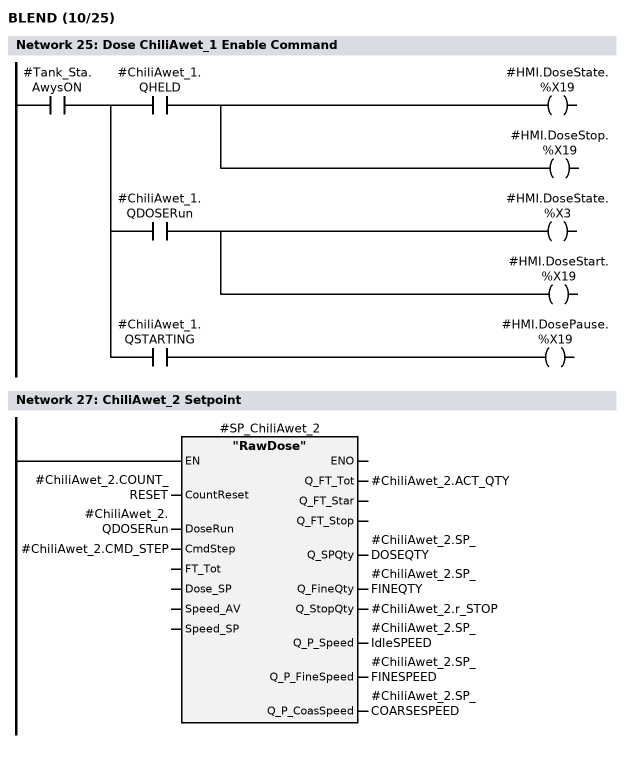
   RUNG wire#powerrail
      Contact( #Tank_Sta.AwysON )
      wire#w1
      Contact( #ChiliAwet_1.QHELD )
      wire#w2
      Coil( #HMI.DoseState.%X19 )
   END_RUNG
   RUNG wire#w2
      Coil( #HMI.DoseStop.%X19 )
   END_RUNG
   RUNG wire#w1
      Contact( #ChiliAwet_1.QDOSERun )
      wire#w3
      Coil( #HMI.DoseState.%X3 )
   END_RUNG
   RUNG wire#w3
      Coil( #HMI.DoseStart.%X19 )
   END_RUNG
   RUNG wire#w1
      Contact( #ChiliAwet_1.QSTARTING )
      Coil( #HMI.DosePause.%X19 )
   END_RUNG
   // the same network as SCL:
   #HMI.DoseState.%X19 := #Tank_Sta.AwysON AND #ChiliAwet_1.QHELD;
   #HMI.DoseStop.%X19 := #HMI.DoseState.%X19;
   #HMI.DoseState.%X3 := #Tank_Sta.AwysON AND #ChiliAwet_1.QDOSERun;
   #HMI.DoseStart.%X19 := #HMI.DoseState.%X3;
   #HMI.DosePause.%X19 := #Tank_Sta.AwysON AND #ChiliAwet_1.QSTARTING;
END_REGION

REGION Network 27: ChiliAwet_2 Setpoint
   RUNG wire#powerrail
      #SP_ChiliAwet_2(CountReset := #ChiliAwet_2.COUNT_RESET, DoseRun := #ChiliAwet_2.QDOSERun, CmdStep := #ChiliAwet_2.CMD_STEP, FT_Tot :=, Dose_SP :=, Speed_AV :=, Speed_SP :=, Q_FT_Tot => #ChiliAwet_2.ACT_QTY, Q_FT_Star =>, Q_FT_Stop =>, Q_SPQty => #ChiliAwet_2.SP_DOSEQTY, Q_FineQty => #ChiliAwet_2.SP_FINEQTY, Q_StopQty => #ChiliAwet_2.r_STOP, Q_P_Speed => #ChiliAwet_2.SP_IdleSPEED, Q_P_FineSpeed => #ChiliAwet_2.SP_FINESPEED, Q_P_CoasSpeed => #ChiliAwet_2.SP_COARSESPEED)
   END_RUNG
   // the same network as SCL:
   #SP_ChiliAwet_2(CountReset := #ChiliAwet_2.COUNT_RESET,   // "RawDose"
                   DoseRun := #ChiliAwet_2.QDOSERun,
                   CmdStep := #ChiliAwet_2.CMD_STEP,
                   Q_FT_Tot => #ChiliAwet_2.ACT_QTY,
                   Q_SPQty => #ChiliAwet_2.SP_DOSEQTY,
                   Q_FineQty => #ChiliAwet_2.SP_FINEQTY,
                   Q_StopQty => #ChiliAwet_2.r_STOP,
                   Q_P_Speed => #ChiliAwet_2.SP_IdleSPEED,
                   Q_P_FineSpeed => #ChiliAwet_2.SP_FINESPEED,
                   Q_P_CoasSpeed => #ChiliAwet_2.SP_COARSESPEED);
END_REGION

REGION Network 28: Dose ChiliAwet_2
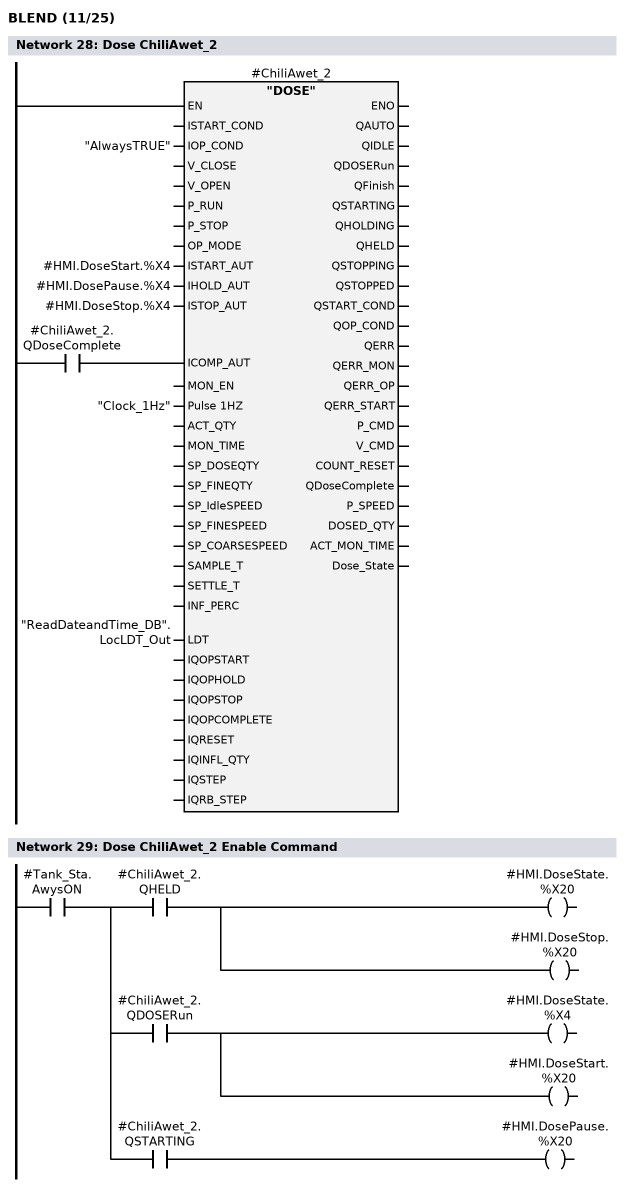
   RUNG wire#powerrail
      #ChiliAwet_2(ICOMP_AUT := wire#w1, ISTART_COND :=, IOP_COND := "AlwaysTRUE", V_CLOSE :=, V_OPEN :=, P_RUN :=, P_STOP :=, OP_MODE :=, ISTART_AUT := #HMI.DoseStart.%X4, IHOLD_AUT := #HMI.DosePause.%X4, ISTOP_AUT := #HMI.DoseStop.%X4, MON_EN :=, "Pulse 1HZ" := "Clock_1Hz", ACT_QTY :=, MON_TIME :=, SP_DOSEQTY :=, SP_FINEQTY :=, SP_IdleSPEED :=, SP_FINESPEED :=, SP_COARSESPEED :=, SAMPLE_T :=, SETTLE_T :=, INF_PERC :=, LDT := "ReadDateandTime_DB".LocLDT_Out, IQOPSTART :=, IQOPHOLD :=, IQOPSTOP :=, IQOPCOMPLETE :=, IQRESET :=, IQINFL_QTY :=, IQSTEP :=, IQRB_STEP :=, QAUTO =>, QIDLE =>, QDOSERun =>, QFinish =>, QSTARTING =>, QHOLDING =>, QHELD =>, QSTOPPING =>, QSTOPPED =>, QSTART_COND =>, QOP_COND =>, QERR =>, QERR_MON =>, QERR_OP =>, QERR_START =>, P_CMD =>, V_CMD =>, COUNT_RESET =>, QDoseComplete =>, P_SPEED =>, DOSED_QTY =>, ACT_MON_TIME =>, Dose_State =>)
   END_RUNG
   RUNG wire#powerrail
      Contact( #ChiliAwet_2.QDoseComplete )
   END_RUNG wire#w1
   // the same network as SCL:
   #ChiliAwet_2(IOP_COND := "AlwaysTRUE",   // "DOSE"
                ISTART_AUT := #HMI.DoseStart.%X4,
                IHOLD_AUT := #HMI.DosePause.%X4,
                ISTOP_AUT := #HMI.DoseStop.%X4,
                ICOMP_AUT := #ChiliAwet_2.QDoseComplete,
                "Pulse 1HZ" := "Clock_1Hz",
                LDT := "ReadDateandTime_DB".LocLDT_Out);
END_REGION

REGION Network 29: Dose ChiliAwet_2 Enable Command
   RUNG wire#powerrail
      Contact( #Tank_Sta.AwysON )
      wire#w1
      Contact( #ChiliAwet_2.QHELD )
      wire#w2
      Coil( #HMI.DoseState.%X20 )
   END_RUNG
   RUNG wire#w2
      Coil( #HMI.DoseStop.%X20 )
   END_RUNG
   RUNG wire#w1
      Contact( #ChiliAwet_2.QDOSERun )
      wire#w3
      Coil( #HMI.DoseState.%X4 )
   END_RUNG
   RUNG wire#w3
      Coil( #HMI.DoseStart.%X20 )
   END_RUNG
   RUNG wire#w1
      Contact( #ChiliAwet_2.QSTARTING )
      Coil( #HMI.DosePause.%X20 )
   END_RUNG
   // the same network as SCL:
   #HMI.DoseState.%X20 := #Tank_Sta.AwysON AND #ChiliAwet_2.QHELD;
   #HMI.DoseStop.%X20 := #HMI.DoseState.%X20;
   #HMI.DoseState.%X4 := #Tank_Sta.AwysON AND #ChiliAwet_2.QDOSERun;
   #HMI.DoseStart.%X20 := #HMI.DoseState.%X4;
   #HMI.DosePause.%X20 := #Tank_Sta.AwysON AND #ChiliAwet_2.QSTARTING;
END_REGION

REGION Network 31: ChiliAwet_3 Setpoint
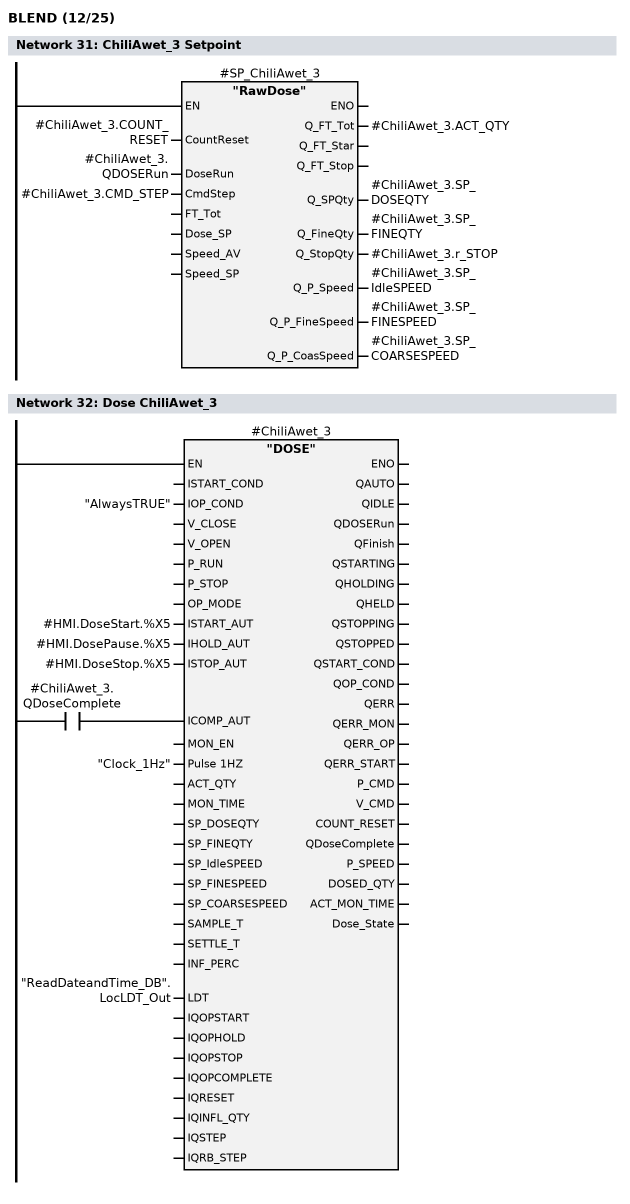
   RUNG wire#powerrail
      #SP_ChiliAwet_3(CountReset := #ChiliAwet_3.COUNT_RESET, DoseRun := #ChiliAwet_3.QDOSERun, CmdStep := #ChiliAwet_3.CMD_STEP, FT_Tot :=, Dose_SP :=, Speed_AV :=, Speed_SP :=, Q_FT_Tot => #ChiliAwet_3.ACT_QTY, Q_FT_Star =>, Q_FT_Stop =>, Q_SPQty => #ChiliAwet_3.SP_DOSEQTY, Q_FineQty => #ChiliAwet_3.SP_FINEQTY, Q_StopQty => #ChiliAwet_3.r_STOP, Q_P_Speed => #ChiliAwet_3.SP_IdleSPEED, Q_P_FineSpeed => #ChiliAwet_3.SP_FINESPEED, Q_P_CoasSpeed => #ChiliAwet_3.SP_COARSESPEED)
   END_RUNG
   // the same network as SCL:
   #SP_ChiliAwet_3(CountReset := #ChiliAwet_3.COUNT_RESET,   // "RawDose"
                   DoseRun := #ChiliAwet_3.QDOSERun,
                   CmdStep := #ChiliAwet_3.CMD_STEP,
                   Q_FT_Tot => #ChiliAwet_3.ACT_QTY,
                   Q_SPQty => #ChiliAwet_3.SP_DOSEQTY,
                   Q_FineQty => #ChiliAwet_3.SP_FINEQTY,
                   Q_StopQty => #ChiliAwet_3.r_STOP,
                   Q_P_Speed => #ChiliAwet_3.SP_IdleSPEED,
                   Q_P_FineSpeed => #ChiliAwet_3.SP_FINESPEED,
                   Q_P_CoasSpeed => #ChiliAwet_3.SP_COARSESPEED);
END_REGION

REGION Network 32: Dose ChiliAwet_3
   RUNG wire#powerrail
      #ChiliAwet_3(ICOMP_AUT := wire#w1, ISTART_COND :=, IOP_COND := "AlwaysTRUE", V_CLOSE :=, V_OPEN :=, P_RUN :=, P_STOP :=, OP_MODE :=, ISTART_AUT := #HMI.DoseStart.%X5, IHOLD_AUT := #HMI.DosePause.%X5, ISTOP_AUT := #HMI.DoseStop.%X5, MON_EN :=, "Pulse 1HZ" := "Clock_1Hz", ACT_QTY :=, MON_TIME :=, SP_DOSEQTY :=, SP_FINEQTY :=, SP_IdleSPEED :=, SP_FINESPEED :=, SP_COARSESPEED :=, SAMPLE_T :=, SETTLE_T :=, INF_PERC :=, LDT := "ReadDateandTime_DB".LocLDT_Out, IQOPSTART :=, IQOPHOLD :=, IQOPSTOP :=, IQOPCOMPLETE :=, IQRESET :=, IQINFL_QTY :=, IQSTEP :=, IQRB_STEP :=, QAUTO =>, QIDLE =>, QDOSERun =>, QFinish =>, QSTARTING =>, QHOLDING =>, QHELD =>, QSTOPPING =>, QSTOPPED =>, QSTART_COND =>, QOP_COND =>, QERR =>, QERR_MON =>, QERR_OP =>, QERR_START =>, P_CMD =>, V_CMD =>, COUNT_RESET =>, QDoseComplete =>, P_SPEED =>, DOSED_QTY =>, ACT_MON_TIME =>, Dose_State =>)
   END_RUNG
   RUNG wire#powerrail
      Contact( #ChiliAwet_3.QDoseComplete )
   END_RUNG wire#w1
   // the same network as SCL:
   #ChiliAwet_3(IOP_COND := "AlwaysTRUE",   // "DOSE"
                ISTART_AUT := #HMI.DoseStart.%X5,
                IHOLD_AUT := #HMI.DosePause.%X5,
                ISTOP_AUT := #HMI.DoseStop.%X5,
                ICOMP_AUT := #ChiliAwet_3.QDoseComplete,
                "Pulse 1HZ" := "Clock_1Hz",
                LDT := "ReadDateandTime_DB".LocLDT_Out);
END_REGION

REGION Network 33: Dose ChiliAwet_3 Enable Command
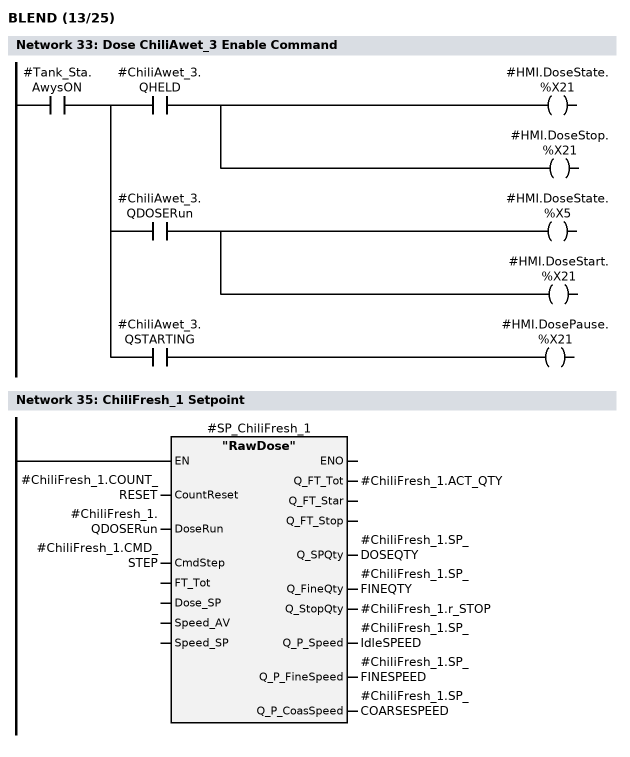
   RUNG wire#powerrail
      Contact( #Tank_Sta.AwysON )
      wire#w1
      Contact( #ChiliAwet_3.QHELD )
      wire#w2
      Coil( #HMI.DoseState.%X21 )
   END_RUNG
   RUNG wire#w2
      Coil( #HMI.DoseStop.%X21 )
   END_RUNG
   RUNG wire#w1
      Contact( #ChiliAwet_3.QDOSERun )
      wire#w3
      Coil( #HMI.DoseState.%X5 )
   END_RUNG
   RUNG wire#w3
      Coil( #HMI.DoseStart.%X21 )
   END_RUNG
   RUNG wire#w1
      Contact( #ChiliAwet_3.QSTARTING )
      Coil( #HMI.DosePause.%X21 )
   END_RUNG
   // the same network as SCL:
   #HMI.DoseState.%X21 := #Tank_Sta.AwysON AND #ChiliAwet_3.QHELD;
   #HMI.DoseStop.%X21 := #HMI.DoseState.%X21;
   #HMI.DoseState.%X5 := #Tank_Sta.AwysON AND #ChiliAwet_3.QDOSERun;
   #HMI.DoseStart.%X21 := #HMI.DoseState.%X5;
   #HMI.DosePause.%X21 := #Tank_Sta.AwysON AND #ChiliAwet_3.QSTARTING;
END_REGION

REGION Network 35: ChiliFresh_1 Setpoint
   RUNG wire#powerrail
      #SP_ChiliFresh_1(CountReset := #ChiliFresh_1.COUNT_RESET, DoseRun := #ChiliFresh_1.QDOSERun, CmdStep := #ChiliFresh_1.CMD_STEP, FT_Tot :=, Dose_SP :=, Speed_AV :=, Speed_SP :=, Q_FT_Tot => #ChiliFresh_1.ACT_QTY, Q_FT_Star =>, Q_FT_Stop =>, Q_SPQty => #ChiliFresh_1.SP_DOSEQTY, Q_FineQty => #ChiliFresh_1.SP_FINEQTY, Q_StopQty => #ChiliFresh_1.r_STOP, Q_P_Speed => #ChiliFresh_1.SP_IdleSPEED, Q_P_FineSpeed => #ChiliFresh_1.SP_FINESPEED, Q_P_CoasSpeed => #ChiliFresh_1.SP_COARSESPEED)
   END_RUNG
   // the same network as SCL:
   #SP_ChiliFresh_1(CountReset := #ChiliFresh_1.COUNT_RESET,   // "RawDose"
                    DoseRun := #ChiliFresh_1.QDOSERun,
                    CmdStep := #ChiliFresh_1.CMD_STEP,
                    Q_FT_Tot => #ChiliFresh_1.ACT_QTY,
                    Q_SPQty => #ChiliFresh_1.SP_DOSEQTY,
                    Q_FineQty => #ChiliFresh_1.SP_FINEQTY,
                    Q_StopQty => #ChiliFresh_1.r_STOP,
                    Q_P_Speed => #ChiliFresh_1.SP_IdleSPEED,
                    Q_P_FineSpeed => #ChiliFresh_1.SP_FINESPEED,
                    Q_P_CoasSpeed => #ChiliFresh_1.SP_COARSESPEED);
END_REGION

REGION Network 36: Dose ChiliFresh_1
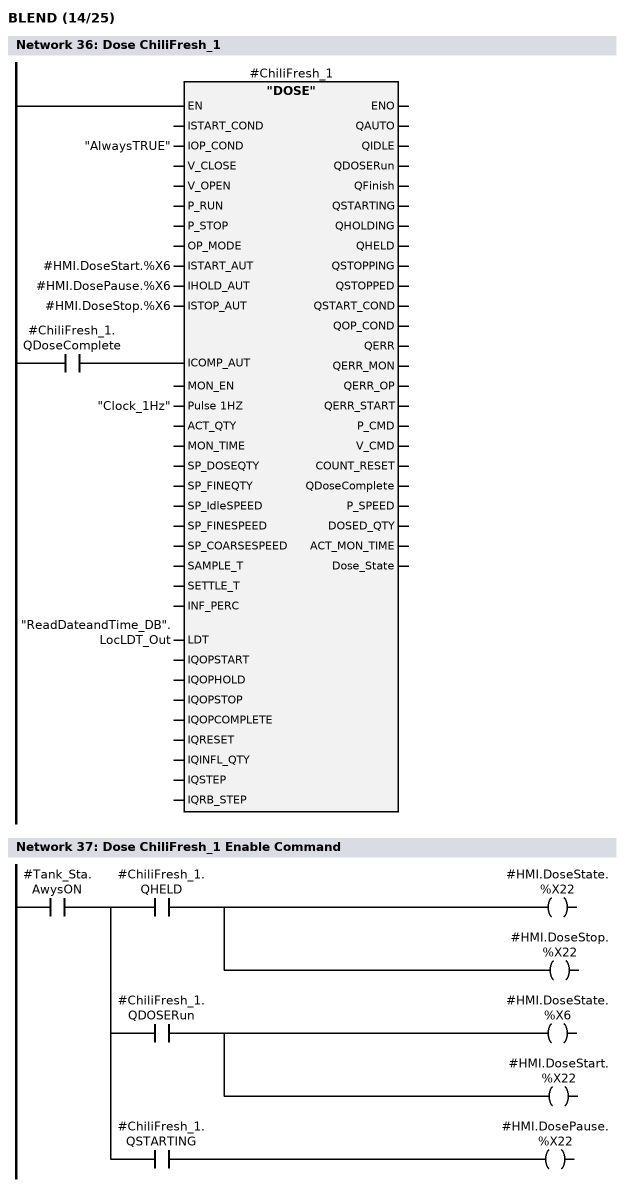
   RUNG wire#powerrail
      #ChiliFresh_1(ICOMP_AUT := wire#w1, ISTART_COND :=, IOP_COND := "AlwaysTRUE", V_CLOSE :=, V_OPEN :=, P_RUN :=, P_STOP :=, OP_MODE :=, ISTART_AUT := #HMI.DoseStart.%X6, IHOLD_AUT := #HMI.DosePause.%X6, ISTOP_AUT := #HMI.DoseStop.%X6, MON_EN :=, "Pulse 1HZ" := "Clock_1Hz", ACT_QTY :=, MON_TIME :=, SP_DOSEQTY :=, SP_FINEQTY :=, SP_IdleSPEED :=, SP_FINESPEED :=, SP_COARSESPEED :=, SAMPLE_T :=, SETTLE_T :=, INF_PERC :=, LDT := "ReadDateandTime_DB".LocLDT_Out, IQOPSTART :=, IQOPHOLD :=, IQOPSTOP :=, IQOPCOMPLETE :=, IQRESET :=, IQINFL_QTY :=, IQSTEP :=, IQRB_STEP :=, QAUTO =>, QIDLE =>, QDOSERun =>, QFinish =>, QSTARTING =>, QHOLDING =>, QHELD =>, QSTOPPING =>, QSTOPPED =>, QSTART_COND =>, QOP_COND =>, QERR =>, QERR_MON =>, QERR_OP =>, QERR_START =>, P_CMD =>, V_CMD =>, COUNT_RESET =>, QDoseComplete =>, P_SPEED =>, DOSED_QTY =>, ACT_MON_TIME =>, Dose_State =>)
   END_RUNG
   RUNG wire#powerrail
      Contact( #ChiliFresh_1.QDoseComplete )
   END_RUNG wire#w1
   // the same network as SCL:
   #ChiliFresh_1(IOP_COND := "AlwaysTRUE",   // "DOSE"
                 ISTART_AUT := #HMI.DoseStart.%X6,
                 IHOLD_AUT := #HMI.DosePause.%X6,
                 ISTOP_AUT := #HMI.DoseStop.%X6,
                 ICOMP_AUT := #ChiliFresh_1.QDoseComplete,
                 "Pulse 1HZ" := "Clock_1Hz",
                 LDT := "ReadDateandTime_DB".LocLDT_Out);
END_REGION

REGION Network 37: Dose ChiliFresh_1 Enable Command
   RUNG wire#powerrail
      Contact( #Tank_Sta.AwysON )
      wire#w1
      Contact( #ChiliFresh_1.QHELD )
      wire#w2
      Coil( #HMI.DoseState.%X22 )
   END_RUNG
   RUNG wire#w2
      Coil( #HMI.DoseStop.%X22 )
   END_RUNG
   RUNG wire#w1
      Contact( #ChiliFresh_1.QDOSERun )
      wire#w3
      Coil( #HMI.DoseState.%X6 )
   END_RUNG
   RUNG wire#w3
      Coil( #HMI.DoseStart.%X22 )
   END_RUNG
   RUNG wire#w1
      Contact( #ChiliFresh_1.QSTARTING )
      Coil( #HMI.DosePause.%X22 )
   END_RUNG
   // the same network as SCL:
   #HMI.DoseState.%X22 := #Tank_Sta.AwysON AND #ChiliFresh_1.QHELD;
   #HMI.DoseStop.%X22 := #HMI.DoseState.%X22;
   #HMI.DoseState.%X6 := #Tank_Sta.AwysON AND #ChiliFresh_1.QDOSERun;
   #HMI.DoseStart.%X22 := #HMI.DoseState.%X6;
   #HMI.DosePause.%X22 := #Tank_Sta.AwysON AND #ChiliFresh_1.QSTARTING;
END_REGION

REGION Network 39: ChiliFresh_2 Setpoint
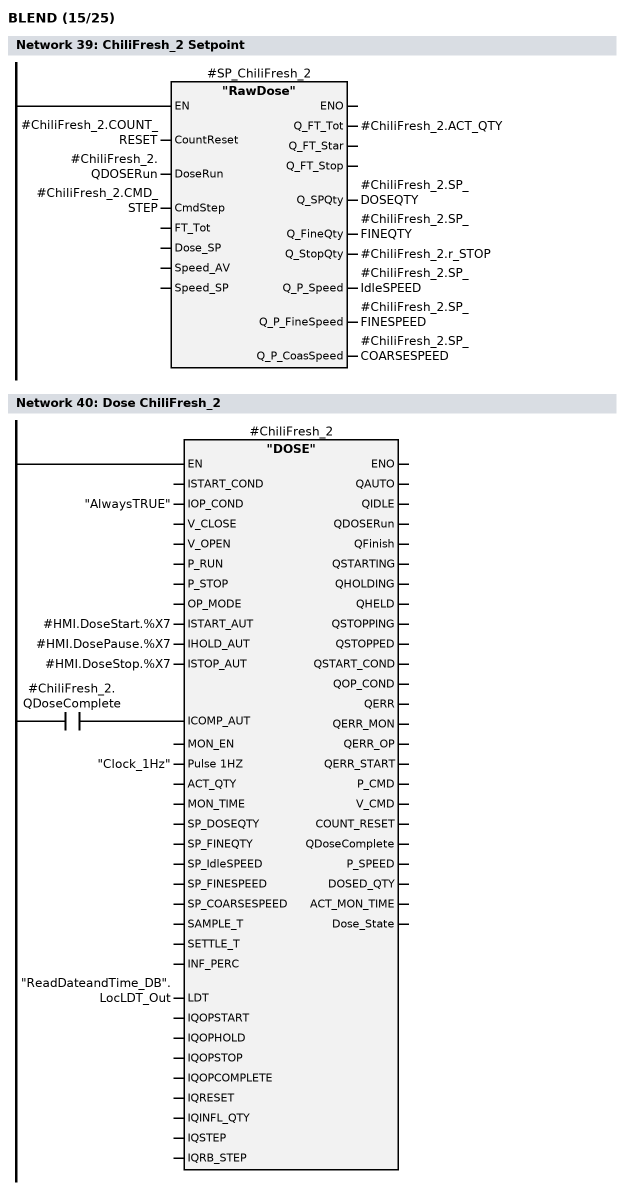
   RUNG wire#powerrail
      #SP_ChiliFresh_2(CountReset := #ChiliFresh_2.COUNT_RESET, DoseRun := #ChiliFresh_2.QDOSERun, CmdStep := #ChiliFresh_2.CMD_STEP, FT_Tot :=, Dose_SP :=, Speed_AV :=, Speed_SP :=, Q_FT_Tot => #ChiliFresh_2.ACT_QTY, Q_FT_Star =>, Q_FT_Stop =>, Q_SPQty => #ChiliFresh_2.SP_DOSEQTY, Q_FineQty => #ChiliFresh_2.SP_FINEQTY, Q_StopQty => #ChiliFresh_2.r_STOP, Q_P_Speed => #ChiliFresh_2.SP_IdleSPEED, Q_P_FineSpeed => #ChiliFresh_2.SP_FINESPEED, Q_P_CoasSpeed => #ChiliFresh_2.SP_COARSESPEED)
   END_RUNG
   // the same network as SCL:
   #SP_ChiliFresh_2(CountReset := #ChiliFresh_2.COUNT_RESET,   // "RawDose"
                    DoseRun := #ChiliFresh_2.QDOSERun,
                    CmdStep := #ChiliFresh_2.CMD_STEP,
                    Q_FT_Tot => #ChiliFresh_2.ACT_QTY,
                    Q_SPQty => #ChiliFresh_2.SP_DOSEQTY,
                    Q_FineQty => #ChiliFresh_2.SP_FINEQTY,
                    Q_StopQty => #ChiliFresh_2.r_STOP,
                    Q_P_Speed => #ChiliFresh_2.SP_IdleSPEED,
                    Q_P_FineSpeed => #ChiliFresh_2.SP_FINESPEED,
                    Q_P_CoasSpeed => #ChiliFresh_2.SP_COARSESPEED);
END_REGION

REGION Network 40: Dose ChiliFresh_2
   RUNG wire#powerrail
      #ChiliFresh_2(ICOMP_AUT := wire#w1, ISTART_COND :=, IOP_COND := "AlwaysTRUE", V_CLOSE :=, V_OPEN :=, P_RUN :=, P_STOP :=, OP_MODE :=, ISTART_AUT := #HMI.DoseStart.%X7, IHOLD_AUT := #HMI.DosePause.%X7, ISTOP_AUT := #HMI.DoseStop.%X7, MON_EN :=, "Pulse 1HZ" := "Clock_1Hz", ACT_QTY :=, MON_TIME :=, SP_DOSEQTY :=, SP_FINEQTY :=, SP_IdleSPEED :=, SP_FINESPEED :=, SP_COARSESPEED :=, SAMPLE_T :=, SETTLE_T :=, INF_PERC :=, LDT := "ReadDateandTime_DB".LocLDT_Out, IQOPSTART :=, IQOPHOLD :=, IQOPSTOP :=, IQOPCOMPLETE :=, IQRESET :=, IQINFL_QTY :=, IQSTEP :=, IQRB_STEP :=, QAUTO =>, QIDLE =>, QDOSERun =>, QFinish =>, QSTARTING =>, QHOLDING =>, QHELD =>, QSTOPPING =>, QSTOPPED =>, QSTART_COND =>, QOP_COND =>, QERR =>, QERR_MON =>, QERR_OP =>, QERR_START =>, P_CMD =>, V_CMD =>, COUNT_RESET =>, QDoseComplete =>, P_SPEED =>, DOSED_QTY =>, ACT_MON_TIME =>, Dose_State =>)
   END_RUNG
   RUNG wire#powerrail
      Contact( #ChiliFresh_2.QDoseComplete )
   END_RUNG wire#w1
   // the same network as SCL:
   #ChiliFresh_2(IOP_COND := "AlwaysTRUE",   // "DOSE"
                 ISTART_AUT := #HMI.DoseStart.%X7,
                 IHOLD_AUT := #HMI.DosePause.%X7,
                 ISTOP_AUT := #HMI.DoseStop.%X7,
                 ICOMP_AUT := #ChiliFresh_2.QDoseComplete,
                 "Pulse 1HZ" := "Clock_1Hz",
                 LDT := "ReadDateandTime_DB".LocLDT_Out);
END_REGION

REGION Network 41: Dose ChiliFresh_2 Enable Command
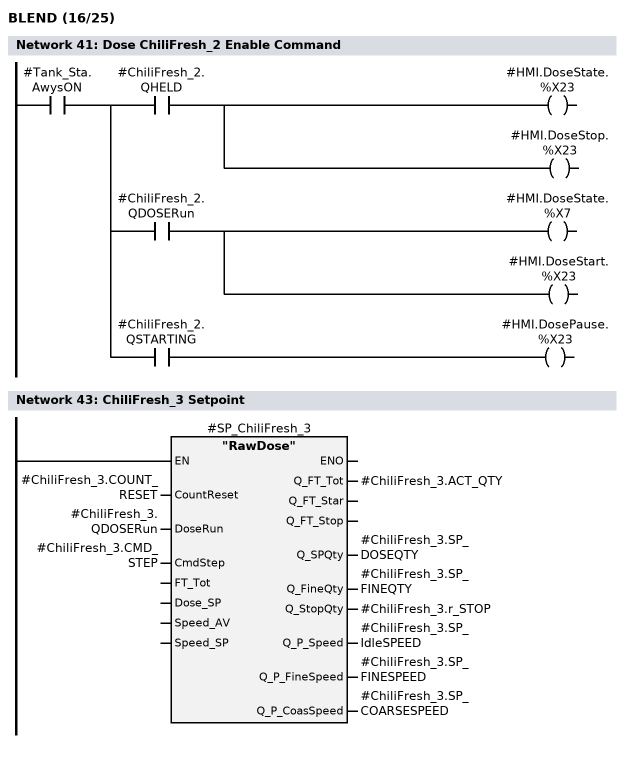
   RUNG wire#powerrail
      Contact( #Tank_Sta.AwysON )
      wire#w1
      Contact( #ChiliFresh_2.QHELD )
      wire#w2
      Coil( #HMI.DoseState.%X23 )
   END_RUNG
   RUNG wire#w2
      Coil( #HMI.DoseStop.%X23 )
   END_RUNG
   RUNG wire#w1
      Contact( #ChiliFresh_2.QDOSERun )
      wire#w3
      Coil( #HMI.DoseState.%X7 )
   END_RUNG
   RUNG wire#w3
      Coil( #HMI.DoseStart.%X23 )
   END_RUNG
   RUNG wire#w1
      Contact( #ChiliFresh_2.QSTARTING )
      Coil( #HMI.DosePause.%X23 )
   END_RUNG
   // the same network as SCL:
   #HMI.DoseState.%X23 := #Tank_Sta.AwysON AND #ChiliFresh_2.QHELD;
   #HMI.DoseStop.%X23 := #HMI.DoseState.%X23;
   #HMI.DoseState.%X7 := #Tank_Sta.AwysON AND #ChiliFresh_2.QDOSERun;
   #HMI.DoseStart.%X23 := #HMI.DoseState.%X7;
   #HMI.DosePause.%X23 := #Tank_Sta.AwysON AND #ChiliFresh_2.QSTARTING;
END_REGION

REGION Network 43: ChiliFresh_3 Setpoint
   RUNG wire#powerrail
      #SP_ChiliFresh_3(CountReset := #ChiliFresh_3.COUNT_RESET, DoseRun := #ChiliFresh_3.QDOSERun, CmdStep := #ChiliFresh_3.CMD_STEP, FT_Tot :=, Dose_SP :=, Speed_AV :=, Speed_SP :=, Q_FT_Tot => #ChiliFresh_3.ACT_QTY, Q_FT_Star =>, Q_FT_Stop =>, Q_SPQty => #ChiliFresh_3.SP_DOSEQTY, Q_FineQty => #ChiliFresh_3.SP_FINEQTY, Q_StopQty => #ChiliFresh_3.r_STOP, Q_P_Speed => #ChiliFresh_3.SP_IdleSPEED, Q_P_FineSpeed => #ChiliFresh_3.SP_FINESPEED, Q_P_CoasSpeed => #ChiliFresh_3.SP_COARSESPEED)
   END_RUNG
   // the same network as SCL:
   #SP_ChiliFresh_3(CountReset := #ChiliFresh_3.COUNT_RESET,   // "RawDose"
                    DoseRun := #ChiliFresh_3.QDOSERun,
                    CmdStep := #ChiliFresh_3.CMD_STEP,
                    Q_FT_Tot => #ChiliFresh_3.ACT_QTY,
                    Q_SPQty => #ChiliFresh_3.SP_DOSEQTY,
                    Q_FineQty => #ChiliFresh_3.SP_FINEQTY,
                    Q_StopQty => #ChiliFresh_3.r_STOP,
                    Q_P_Speed => #ChiliFresh_3.SP_IdleSPEED,
                    Q_P_FineSpeed => #ChiliFresh_3.SP_FINESPEED,
                    Q_P_CoasSpeed => #ChiliFresh_3.SP_COARSESPEED);
END_REGION

REGION Network 44: Dose ChiliFresh_3
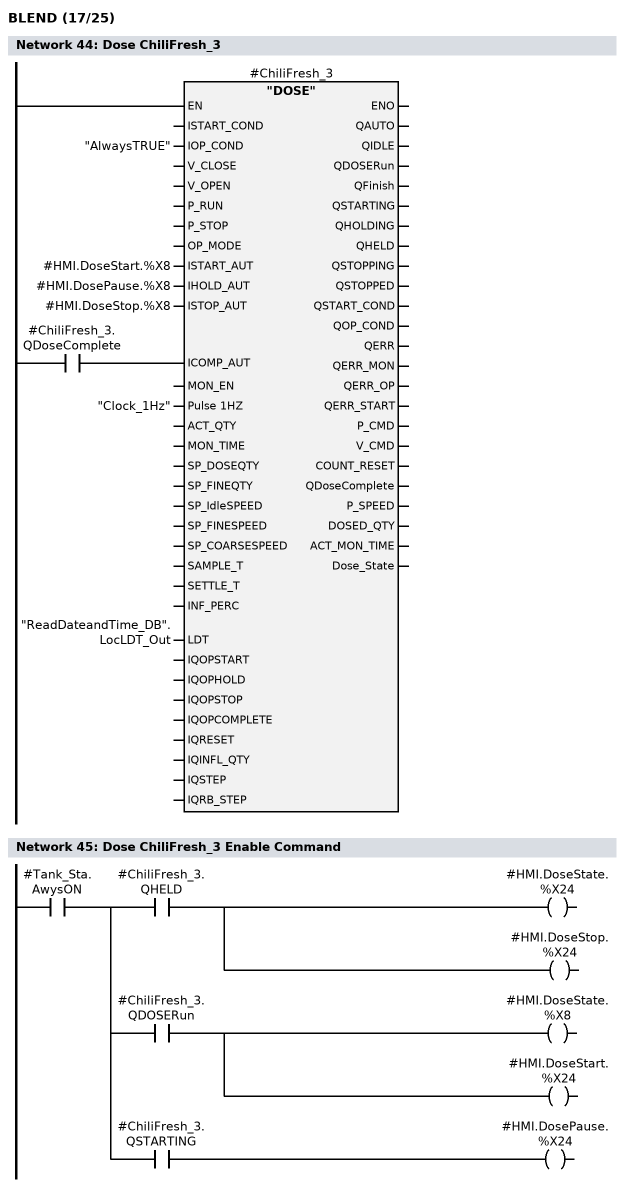
   RUNG wire#powerrail
      #ChiliFresh_3(ICOMP_AUT := wire#w1, ISTART_COND :=, IOP_COND := "AlwaysTRUE", V_CLOSE :=, V_OPEN :=, P_RUN :=, P_STOP :=, OP_MODE :=, ISTART_AUT := #HMI.DoseStart.%X8, IHOLD_AUT := #HMI.DosePause.%X8, ISTOP_AUT := #HMI.DoseStop.%X8, MON_EN :=, "Pulse 1HZ" := "Clock_1Hz", ACT_QTY :=, MON_TIME :=, SP_DOSEQTY :=, SP_FINEQTY :=, SP_IdleSPEED :=, SP_FINESPEED :=, SP_COARSESPEED :=, SAMPLE_T :=, SETTLE_T :=, INF_PERC :=, LDT := "ReadDateandTime_DB".LocLDT_Out, IQOPSTART :=, IQOPHOLD :=, IQOPSTOP :=, IQOPCOMPLETE :=, IQRESET :=, IQINFL_QTY :=, IQSTEP :=, IQRB_STEP :=, QAUTO =>, QIDLE =>, QDOSERun =>, QFinish =>, QSTARTING =>, QHOLDING =>, QHELD =>, QSTOPPING =>, QSTOPPED =>, QSTART_COND =>, QOP_COND =>, QERR =>, QERR_MON =>, QERR_OP =>, QERR_START =>, P_CMD =>, V_CMD =>, COUNT_RESET =>, QDoseComplete =>, P_SPEED =>, DOSED_QTY =>, ACT_MON_TIME =>, Dose_State =>)
   END_RUNG
   RUNG wire#powerrail
      Contact( #ChiliFresh_3.QDoseComplete )
   END_RUNG wire#w1
   // the same network as SCL:
   #ChiliFresh_3(IOP_COND := "AlwaysTRUE",   // "DOSE"
                 ISTART_AUT := #HMI.DoseStart.%X8,
                 IHOLD_AUT := #HMI.DosePause.%X8,
                 ISTOP_AUT := #HMI.DoseStop.%X8,
                 ICOMP_AUT := #ChiliFresh_3.QDoseComplete,
                 "Pulse 1HZ" := "Clock_1Hz",
                 LDT := "ReadDateandTime_DB".LocLDT_Out);
END_REGION

REGION Network 45: Dose ChiliFresh_3 Enable Command
   RUNG wire#powerrail
      Contact( #Tank_Sta.AwysON )
      wire#w1
      Contact( #ChiliFresh_3.QHELD )
      wire#w2
      Coil( #HMI.DoseState.%X24 )
   END_RUNG
   RUNG wire#w2
      Coil( #HMI.DoseStop.%X24 )
   END_RUNG
   RUNG wire#w1
      Contact( #ChiliFresh_3.QDOSERun )
      wire#w3
      Coil( #HMI.DoseState.%X8 )
   END_RUNG
   RUNG wire#w3
      Coil( #HMI.DoseStart.%X24 )
   END_RUNG
   RUNG wire#w1
      Contact( #ChiliFresh_3.QSTARTING )
      Coil( #HMI.DosePause.%X24 )
   END_RUNG
   // the same network as SCL:
   #HMI.DoseState.%X24 := #Tank_Sta.AwysON AND #ChiliFresh_3.QHELD;
   #HMI.DoseStop.%X24 := #HMI.DoseState.%X24;
   #HMI.DoseState.%X8 := #Tank_Sta.AwysON AND #ChiliFresh_3.QDOSERun;
   #HMI.DoseStart.%X24 := #HMI.DoseState.%X8;
   #HMI.DosePause.%X24 := #Tank_Sta.AwysON AND #ChiliFresh_3.QSTARTING;
END_REGION

REGION Network 47: Garlic Setpoint
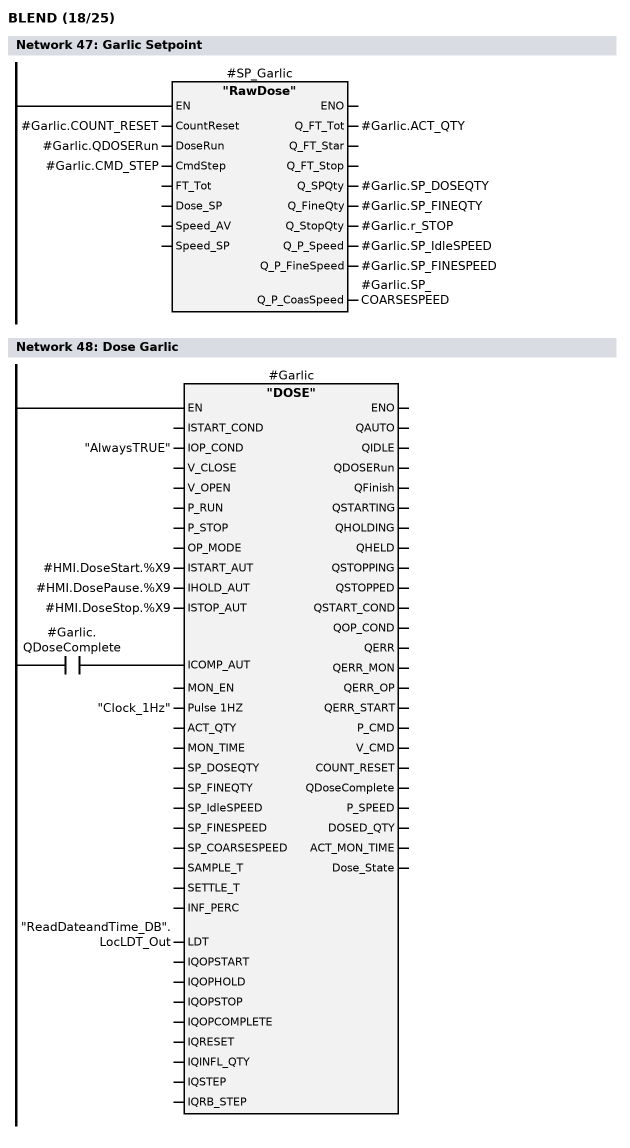
   RUNG wire#powerrail
      #SP_Garlic(CountReset := #Garlic.COUNT_RESET, DoseRun := #Garlic.QDOSERun, CmdStep := #Garlic.CMD_STEP, FT_Tot :=, Dose_SP :=, Speed_AV :=, Speed_SP :=, Q_FT_Tot => #Garlic.ACT_QTY, Q_FT_Star =>, Q_FT_Stop =>, Q_SPQty => #Garlic.SP_DOSEQTY, Q_FineQty => #Garlic.SP_FINEQTY, Q_StopQty => #Garlic.r_STOP, Q_P_Speed => #Garlic.SP_IdleSPEED, Q_P_FineSpeed => #Garlic.SP_FINESPEED, Q_P_CoasSpeed => #Garlic.SP_COARSESPEED)
   END_RUNG
   // the same network as SCL:
   #SP_Garlic(CountReset := #Garlic.COUNT_RESET,   // "RawDose"
              DoseRun := #Garlic.QDOSERun,
              CmdStep := #Garlic.CMD_STEP,
              Q_FT_Tot => #Garlic.ACT_QTY,
              Q_SPQty => #Garlic.SP_DOSEQTY,
              Q_FineQty => #Garlic.SP_FINEQTY,
              Q_StopQty => #Garlic.r_STOP,
              Q_P_Speed => #Garlic.SP_IdleSPEED,
              Q_P_FineSpeed => #Garlic.SP_FINESPEED,
              Q_P_CoasSpeed => #Garlic.SP_COARSESPEED);
END_REGION

REGION Network 48: Dose Garlic
   RUNG wire#powerrail
      #Garlic(ICOMP_AUT := wire#w1, ISTART_COND :=, IOP_COND := "AlwaysTRUE", V_CLOSE :=, V_OPEN :=, P_RUN :=, P_STOP :=, OP_MODE :=, ISTART_AUT := #HMI.DoseStart.%X9, IHOLD_AUT := #HMI.DosePause.%X9, ISTOP_AUT := #HMI.DoseStop.%X9, MON_EN :=, "Pulse 1HZ" := "Clock_1Hz", ACT_QTY :=, MON_TIME :=, SP_DOSEQTY :=, SP_FINEQTY :=, SP_IdleSPEED :=, SP_FINESPEED :=, SP_COARSESPEED :=, SAMPLE_T :=, SETTLE_T :=, INF_PERC :=, LDT := "ReadDateandTime_DB".LocLDT_Out, IQOPSTART :=, IQOPHOLD :=, IQOPSTOP :=, IQOPCOMPLETE :=, IQRESET :=, IQINFL_QTY :=, IQSTEP :=, IQRB_STEP :=, QAUTO =>, QIDLE =>, QDOSERun =>, QFinish =>, QSTARTING =>, QHOLDING =>, QHELD =>, QSTOPPING =>, QSTOPPED =>, QSTART_COND =>, QOP_COND =>, QERR =>, QERR_MON =>, QERR_OP =>, QERR_START =>, P_CMD =>, V_CMD =>, COUNT_RESET =>, QDoseComplete =>, P_SPEED =>, DOSED_QTY =>, ACT_MON_TIME =>, Dose_State =>)
   END_RUNG
   RUNG wire#powerrail
      Contact( #Garlic.QDoseComplete )
   END_RUNG wire#w1
   // the same network as SCL:
   #Garlic(IOP_COND := "AlwaysTRUE",   // "DOSE"
           ISTART_AUT := #HMI.DoseStart.%X9,
           IHOLD_AUT := #HMI.DosePause.%X9,
           ISTOP_AUT := #HMI.DoseStop.%X9,
           ICOMP_AUT := #Garlic.QDoseComplete,
           "Pulse 1HZ" := "Clock_1Hz",
           LDT := "ReadDateandTime_DB".LocLDT_Out);
END_REGION

REGION Network 49: Dose Garlic Enable Command
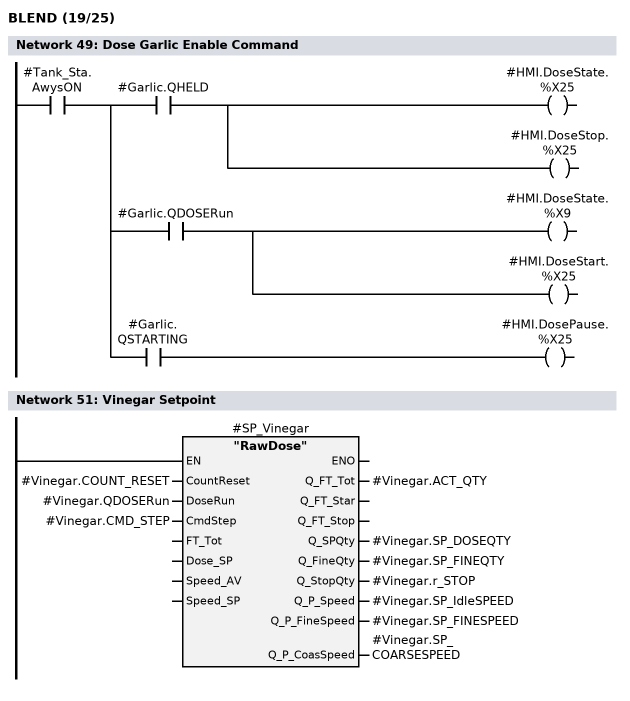
   RUNG wire#powerrail
      Contact( #Tank_Sta.AwysON )
      wire#w1
      Contact( #Garlic.QHELD )
      wire#w2
      Coil( #HMI.DoseState.%X25 )
   END_RUNG
   RUNG wire#w2
      Coil( #HMI.DoseStop.%X25 )
   END_RUNG
   RUNG wire#w1
      Contact( #Garlic.QDOSERun )
      wire#w3
      Coil( #HMI.DoseState.%X9 )
   END_RUNG
   RUNG wire#w3
      Coil( #HMI.DoseStart.%X25 )
   END_RUNG
   RUNG wire#w1
      Contact( #Garlic.QSTARTING )
      Coil( #HMI.DosePause.%X25 )
   END_RUNG
   // the same network as SCL:
   #HMI.DoseState.%X25 := #Tank_Sta.AwysON AND #Garlic.QHELD;
   #HMI.DoseStop.%X25 := #HMI.DoseState.%X25;
   #HMI.DoseState.%X9 := #Tank_Sta.AwysON AND #Garlic.QDOSERun;
   #HMI.DoseStart.%X25 := #HMI.DoseState.%X9;
   #HMI.DosePause.%X25 := #Tank_Sta.AwysON AND #Garlic.QSTARTING;
END_REGION

REGION Network 51: Vinegar Setpoint
   RUNG wire#powerrail
      #SP_Vinegar(CountReset := #Vinegar.COUNT_RESET, DoseRun := #Vinegar.QDOSERun, CmdStep := #Vinegar.CMD_STEP, FT_Tot :=, Dose_SP :=, Speed_AV :=, Speed_SP :=, Q_FT_Tot => #Vinegar.ACT_QTY, Q_FT_Star =>, Q_FT_Stop =>, Q_SPQty => #Vinegar.SP_DOSEQTY, Q_FineQty => #Vinegar.SP_FINEQTY, Q_StopQty => #Vinegar.r_STOP, Q_P_Speed => #Vinegar.SP_IdleSPEED, Q_P_FineSpeed => #Vinegar.SP_FINESPEED, Q_P_CoasSpeed => #Vinegar.SP_COARSESPEED)
   END_RUNG
   // the same network as SCL:
   #SP_Vinegar(CountReset := #Vinegar.COUNT_RESET,   // "RawDose"
               DoseRun := #Vinegar.QDOSERun,
               CmdStep := #Vinegar.CMD_STEP,
               Q_FT_Tot => #Vinegar.ACT_QTY,
               Q_SPQty => #Vinegar.SP_DOSEQTY,
               Q_FineQty => #Vinegar.SP_FINEQTY,
               Q_StopQty => #Vinegar.r_STOP,
               Q_P_Speed => #Vinegar.SP_IdleSPEED,
               Q_P_FineSpeed => #Vinegar.SP_FINESPEED,
               Q_P_CoasSpeed => #Vinegar.SP_COARSESPEED);
END_REGION

REGION Network 52: Dose Vinegar
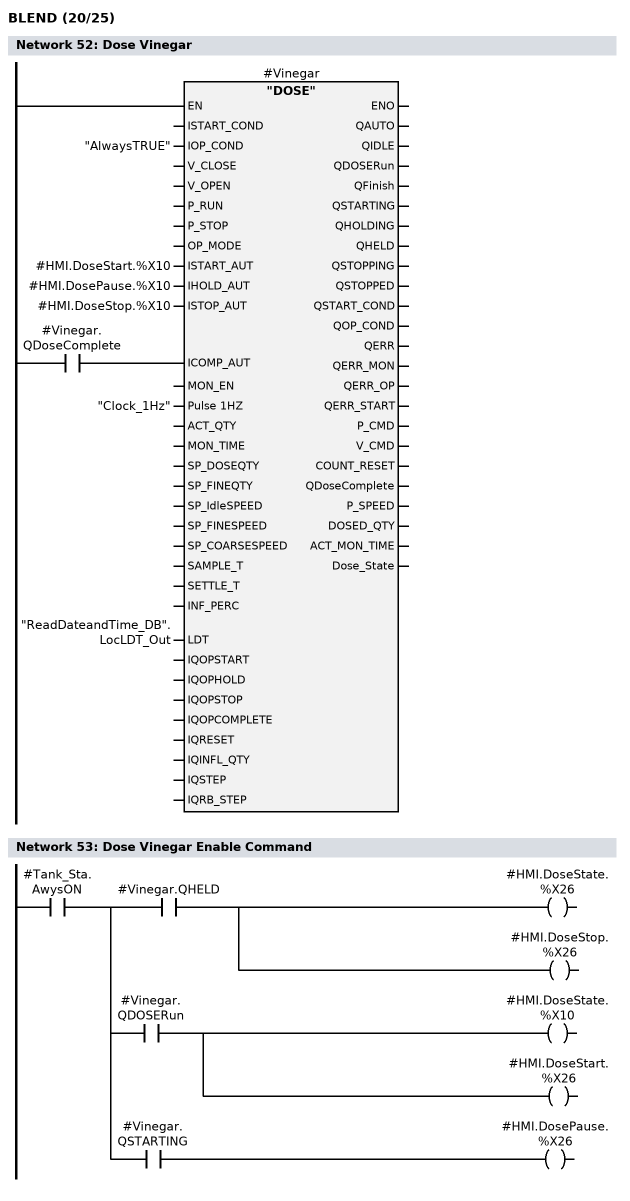
   RUNG wire#powerrail
      #Vinegar(ICOMP_AUT := wire#w1, ISTART_COND :=, IOP_COND := "AlwaysTRUE", V_CLOSE :=, V_OPEN :=, P_RUN :=, P_STOP :=, OP_MODE :=, ISTART_AUT := #HMI.DoseStart.%X10, IHOLD_AUT := #HMI.DosePause.%X10, ISTOP_AUT := #HMI.DoseStop.%X10, MON_EN :=, "Pulse 1HZ" := "Clock_1Hz", ACT_QTY :=, MON_TIME :=, SP_DOSEQTY :=, SP_FINEQTY :=, SP_IdleSPEED :=, SP_FINESPEED :=, SP_COARSESPEED :=, SAMPLE_T :=, SETTLE_T :=, INF_PERC :=, LDT := "ReadDateandTime_DB".LocLDT_Out, IQOPSTART :=, IQOPHOLD :=, IQOPSTOP :=, IQOPCOMPLETE :=, IQRESET :=, IQINFL_QTY :=, IQSTEP :=, IQRB_STEP :=, QAUTO =>, QIDLE =>, QDOSERun =>, QFinish =>, QSTARTING =>, QHOLDING =>, QHELD =>, QSTOPPING =>, QSTOPPED =>, QSTART_COND =>, QOP_COND =>, QERR =>, QERR_MON =>, QERR_OP =>, QERR_START =>, P_CMD =>, V_CMD =>, COUNT_RESET =>, QDoseComplete =>, P_SPEED =>, DOSED_QTY =>, ACT_MON_TIME =>, Dose_State =>)
   END_RUNG
   RUNG wire#powerrail
      Contact( #Vinegar.QDoseComplete )
   END_RUNG wire#w1
   // the same network as SCL:
   #Vinegar(IOP_COND := "AlwaysTRUE",   // "DOSE"
            ISTART_AUT := #HMI.DoseStart.%X10,
            IHOLD_AUT := #HMI.DosePause.%X10,
            ISTOP_AUT := #HMI.DoseStop.%X10,
            ICOMP_AUT := #Vinegar.QDoseComplete,
            "Pulse 1HZ" := "Clock_1Hz",
            LDT := "ReadDateandTime_DB".LocLDT_Out);
END_REGION

REGION Network 53: Dose Vinegar Enable Command
   RUNG wire#powerrail
      Contact( #Tank_Sta.AwysON )
      wire#w1
      Contact( #Vinegar.QHELD )
      wire#w2
      Coil( #HMI.DoseState.%X26 )
   END_RUNG
   RUNG wire#w2
      Coil( #HMI.DoseStop.%X26 )
   END_RUNG
   RUNG wire#w1
      Contact( #Vinegar.QDOSERun )
      wire#w3
      Coil( #HMI.DoseState.%X10 )
   END_RUNG
   RUNG wire#w3
      Coil( #HMI.DoseStart.%X26 )
   END_RUNG
   RUNG wire#w1
      Contact( #Vinegar.QSTARTING )
      Coil( #HMI.DosePause.%X26 )
   END_RUNG
   // the same network as SCL:
   #HMI.DoseState.%X26 := #Tank_Sta.AwysON AND #Vinegar.QHELD;
   #HMI.DoseStop.%X26 := #HMI.DoseState.%X26;
   #HMI.DoseState.%X10 := #Tank_Sta.AwysON AND #Vinegar.QDOSERun;
   #HMI.DoseStart.%X26 := #HMI.DoseState.%X10;
   #HMI.DosePause.%X26 := #Tank_Sta.AwysON AND #Vinegar.QSTARTING;
END_REGION

REGION Network 55: Tomato Setpoint
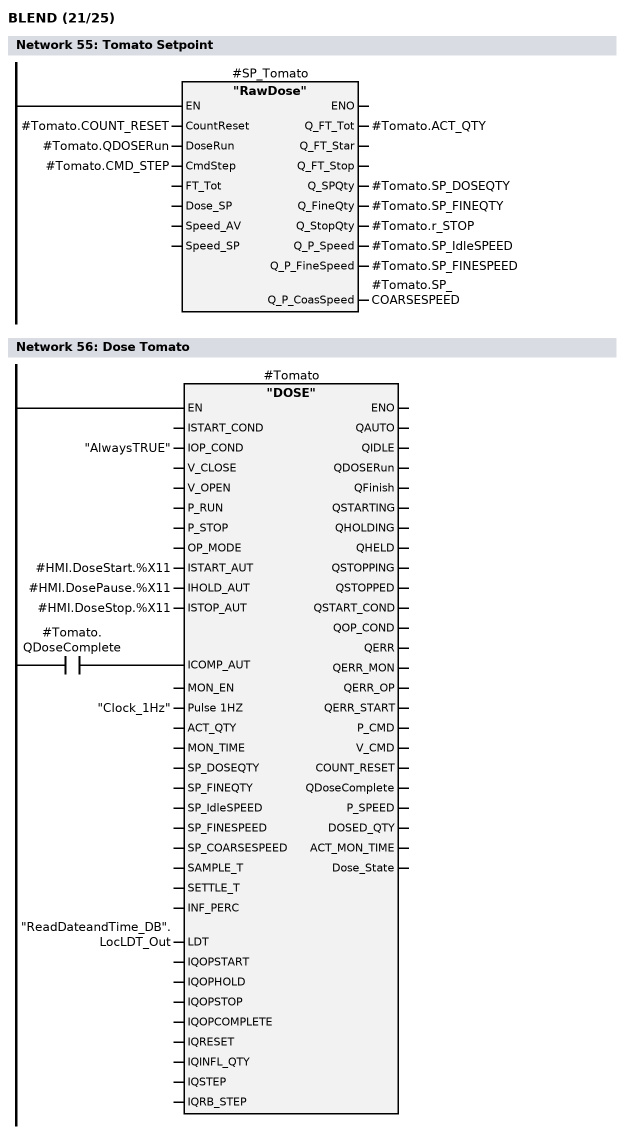
   RUNG wire#powerrail
      #SP_Tomato(CountReset := #Tomato.COUNT_RESET, DoseRun := #Tomato.QDOSERun, CmdStep := #Tomato.CMD_STEP, FT_Tot :=, Dose_SP :=, Speed_AV :=, Speed_SP :=, Q_FT_Tot => #Tomato.ACT_QTY, Q_FT_Star =>, Q_FT_Stop =>, Q_SPQty => #Tomato.SP_DOSEQTY, Q_FineQty => #Tomato.SP_FINEQTY, Q_StopQty => #Tomato.r_STOP, Q_P_Speed => #Tomato.SP_IdleSPEED, Q_P_FineSpeed => #Tomato.SP_FINESPEED, Q_P_CoasSpeed => #Tomato.SP_COARSESPEED)
   END_RUNG
   // the same network as SCL:
   #SP_Tomato(CountReset := #Tomato.COUNT_RESET,   // "RawDose"
              DoseRun := #Tomato.QDOSERun,
              CmdStep := #Tomato.CMD_STEP,
              Q_FT_Tot => #Tomato.ACT_QTY,
              Q_SPQty => #Tomato.SP_DOSEQTY,
              Q_FineQty => #Tomato.SP_FINEQTY,
              Q_StopQty => #Tomato.r_STOP,
              Q_P_Speed => #Tomato.SP_IdleSPEED,
              Q_P_FineSpeed => #Tomato.SP_FINESPEED,
              Q_P_CoasSpeed => #Tomato.SP_COARSESPEED);
END_REGION

REGION Network 56: Dose Tomato
   RUNG wire#powerrail
      #Tomato(ICOMP_AUT := wire#w1, ISTART_COND :=, IOP_COND := "AlwaysTRUE", V_CLOSE :=, V_OPEN :=, P_RUN :=, P_STOP :=, OP_MODE :=, ISTART_AUT := #HMI.DoseStart.%X11, IHOLD_AUT := #HMI.DosePause.%X11, ISTOP_AUT := #HMI.DoseStop.%X11, MON_EN :=, "Pulse 1HZ" := "Clock_1Hz", ACT_QTY :=, MON_TIME :=, SP_DOSEQTY :=, SP_FINEQTY :=, SP_IdleSPEED :=, SP_FINESPEED :=, SP_COARSESPEED :=, SAMPLE_T :=, SETTLE_T :=, INF_PERC :=, LDT := "ReadDateandTime_DB".LocLDT_Out, IQOPSTART :=, IQOPHOLD :=, IQOPSTOP :=, IQOPCOMPLETE :=, IQRESET :=, IQINFL_QTY :=, IQSTEP :=, IQRB_STEP :=, QAUTO =>, QIDLE =>, QDOSERun =>, QFinish =>, QSTARTING =>, QHOLDING =>, QHELD =>, QSTOPPING =>, QSTOPPED =>, QSTART_COND =>, QOP_COND =>, QERR =>, QERR_MON =>, QERR_OP =>, QERR_START =>, P_CMD =>, V_CMD =>, COUNT_RESET =>, QDoseComplete =>, P_SPEED =>, DOSED_QTY =>, ACT_MON_TIME =>, Dose_State =>)
   END_RUNG
   RUNG wire#powerrail
      Contact( #Tomato.QDoseComplete )
   END_RUNG wire#w1
   // the same network as SCL:
   #Tomato(IOP_COND := "AlwaysTRUE",   // "DOSE"
           ISTART_AUT := #HMI.DoseStart.%X11,
           IHOLD_AUT := #HMI.DosePause.%X11,
           ISTOP_AUT := #HMI.DoseStop.%X11,
           ICOMP_AUT := #Tomato.QDoseComplete,
           "Pulse 1HZ" := "Clock_1Hz",
           LDT := "ReadDateandTime_DB".LocLDT_Out);
END_REGION

REGION Network 57: Dose Tomato Enable Command
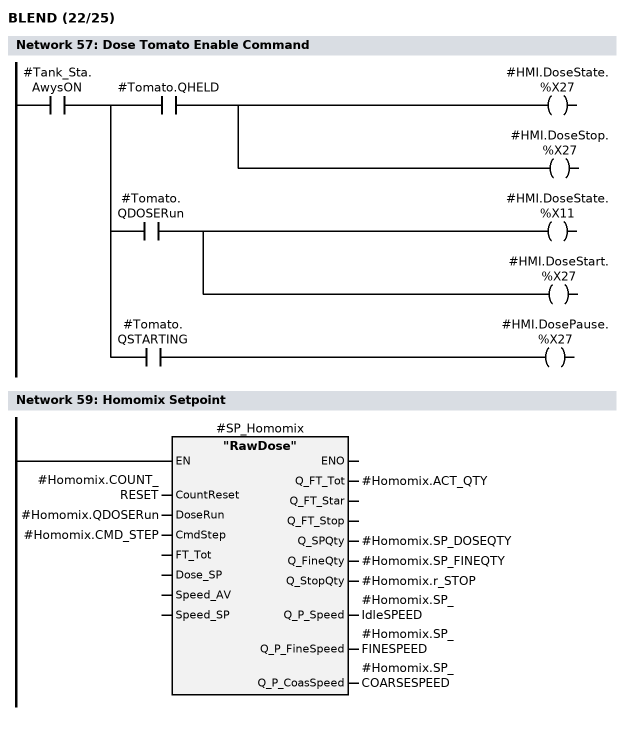
   RUNG wire#powerrail
      Contact( #Tank_Sta.AwysON )
      wire#w1
      Contact( #Tomato.QHELD )
      wire#w2
      Coil( #HMI.DoseState.%X27 )
   END_RUNG
   RUNG wire#w2
      Coil( #HMI.DoseStop.%X27 )
   END_RUNG
   RUNG wire#w1
      Contact( #Tomato.QDOSERun )
      wire#w3
      Coil( #HMI.DoseState.%X11 )
   END_RUNG
   RUNG wire#w3
      Coil( #HMI.DoseStart.%X27 )
   END_RUNG
   RUNG wire#w1
      Contact( #Tomato.QSTARTING )
      Coil( #HMI.DosePause.%X27 )
   END_RUNG
   // the same network as SCL:
   #HMI.DoseState.%X27 := #Tank_Sta.AwysON AND #Tomato.QHELD;
   #HMI.DoseStop.%X27 := #HMI.DoseState.%X27;
   #HMI.DoseState.%X11 := #Tank_Sta.AwysON AND #Tomato.QDOSERun;
   #HMI.DoseStart.%X27 := #HMI.DoseState.%X11;
   #HMI.DosePause.%X27 := #Tank_Sta.AwysON AND #Tomato.QSTARTING;
END_REGION

REGION Network 59: Homomix Setpoint
   RUNG wire#powerrail
      #SP_Homomix(CountReset := #Homomix.COUNT_RESET, DoseRun := #Homomix.QDOSERun, CmdStep := #Homomix.CMD_STEP, FT_Tot :=, Dose_SP :=, Speed_AV :=, Speed_SP :=, Q_FT_Tot => #Homomix.ACT_QTY, Q_FT_Star =>, Q_FT_Stop =>, Q_SPQty => #Homomix.SP_DOSEQTY, Q_FineQty => #Homomix.SP_FINEQTY, Q_StopQty => #Homomix.r_STOP, Q_P_Speed => #Homomix.SP_IdleSPEED, Q_P_FineSpeed => #Homomix.SP_FINESPEED, Q_P_CoasSpeed => #Homomix.SP_COARSESPEED)
   END_RUNG
   // the same network as SCL:
   #SP_Homomix(CountReset := #Homomix.COUNT_RESET,   // "RawDose"
               DoseRun := #Homomix.QDOSERun,
               CmdStep := #Homomix.CMD_STEP,
               Q_FT_Tot => #Homomix.ACT_QTY,
               Q_SPQty => #Homomix.SP_DOSEQTY,
               Q_FineQty => #Homomix.SP_FINEQTY,
               Q_StopQty => #Homomix.r_STOP,
               Q_P_Speed => #Homomix.SP_IdleSPEED,
               Q_P_FineSpeed => #Homomix.SP_FINESPEED,
               Q_P_CoasSpeed => #Homomix.SP_COARSESPEED);
END_REGION

REGION Network 60: Dose Homomix
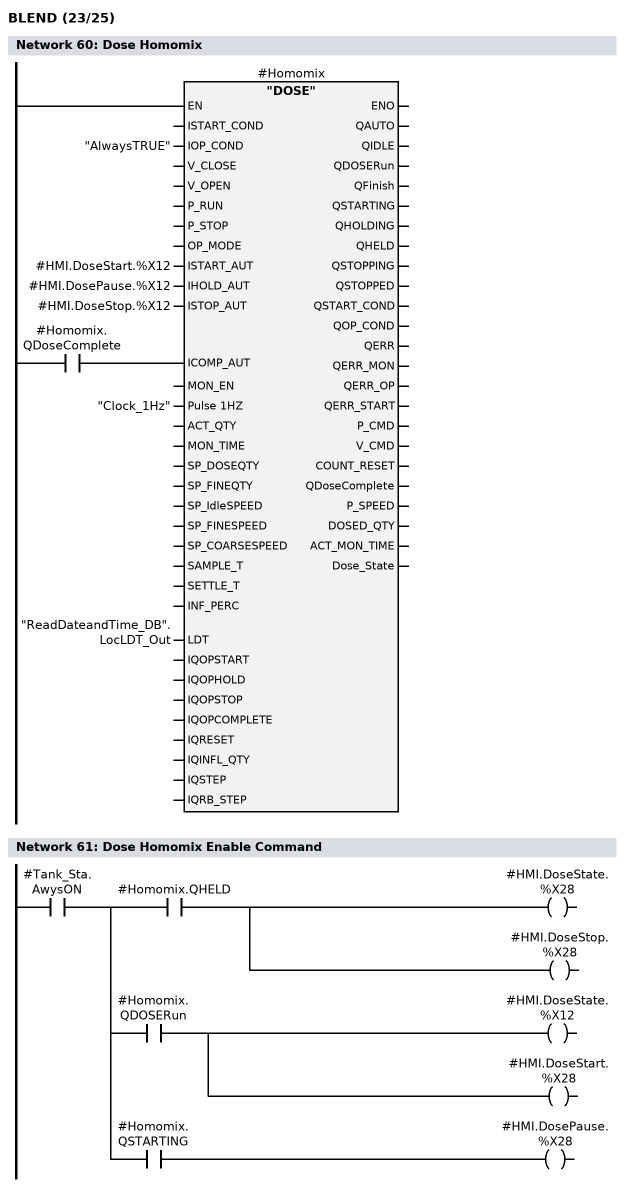
   RUNG wire#powerrail
      #Homomix(ICOMP_AUT := wire#w1, ISTART_COND :=, IOP_COND := "AlwaysTRUE", V_CLOSE :=, V_OPEN :=, P_RUN :=, P_STOP :=, OP_MODE :=, ISTART_AUT := #HMI.DoseStart.%X12, IHOLD_AUT := #HMI.DosePause.%X12, ISTOP_AUT := #HMI.DoseStop.%X12, MON_EN :=, "Pulse 1HZ" := "Clock_1Hz", ACT_QTY :=, MON_TIME :=, SP_DOSEQTY :=, SP_FINEQTY :=, SP_IdleSPEED :=, SP_FINESPEED :=, SP_COARSESPEED :=, SAMPLE_T :=, SETTLE_T :=, INF_PERC :=, LDT := "ReadDateandTime_DB".LocLDT_Out, IQOPSTART :=, IQOPHOLD :=, IQOPSTOP :=, IQOPCOMPLETE :=, IQRESET :=, IQINFL_QTY :=, IQSTEP :=, IQRB_STEP :=, QAUTO =>, QIDLE =>, QDOSERun =>, QFinish =>, QSTARTING =>, QHOLDING =>, QHELD =>, QSTOPPING =>, QSTOPPED =>, QSTART_COND =>, QOP_COND =>, QERR =>, QERR_MON =>, QERR_OP =>, QERR_START =>, P_CMD =>, V_CMD =>, COUNT_RESET =>, QDoseComplete =>, P_SPEED =>, DOSED_QTY =>, ACT_MON_TIME =>, Dose_State =>)
   END_RUNG
   RUNG wire#powerrail
      Contact( #Homomix.QDoseComplete )
   END_RUNG wire#w1
   // the same network as SCL:
   #Homomix(IOP_COND := "AlwaysTRUE",   // "DOSE"
            ISTART_AUT := #HMI.DoseStart.%X12,
            IHOLD_AUT := #HMI.DosePause.%X12,
            ISTOP_AUT := #HMI.DoseStop.%X12,
            ICOMP_AUT := #Homomix.QDoseComplete,
            "Pulse 1HZ" := "Clock_1Hz",
            LDT := "ReadDateandTime_DB".LocLDT_Out);
END_REGION

REGION Network 61: Dose Homomix Enable Command
   RUNG wire#powerrail
      Contact( #Tank_Sta.AwysON )
      wire#w1
      Contact( #Homomix.QHELD )
      wire#w2
      Coil( #HMI.DoseState.%X28 )
   END_RUNG
   RUNG wire#w2
      Coil( #HMI.DoseStop.%X28 )
   END_RUNG
   RUNG wire#w1
      Contact( #Homomix.QDOSERun )
      wire#w3
      Coil( #HMI.DoseState.%X12 )
   END_RUNG
   RUNG wire#w3
      Coil( #HMI.DoseStart.%X28 )
   END_RUNG
   RUNG wire#w1
      Contact( #Homomix.QSTARTING )
      Coil( #HMI.DosePause.%X28 )
   END_RUNG
   // the same network as SCL:
   #HMI.DoseState.%X28 := #Tank_Sta.AwysON AND #Homomix.QHELD;
   #HMI.DoseStop.%X28 := #HMI.DoseState.%X28;
   #HMI.DoseState.%X12 := #Tank_Sta.AwysON AND #Homomix.QDOSERun;
   #HMI.DoseStart.%X28 := #HMI.DoseState.%X12;
   #HMI.DosePause.%X28 := #Tank_Sta.AwysON AND #Homomix.QSTARTING;
END_REGION

REGION Network 63: Rework Setpoint
